  PROC DrawPart36()
    MoveL Offs(pOrigin,159.05,133.27,0.00),v40,z0,tPen\WObj:=wPaper;
    MoveL Offs(pOrigin,159.60,133.02,0.00),v40,z0,tPen\WObj:=wPaper;
    MoveL Offs(pOrigin,155.70,129.11,0.00),v40,z0,tPen\WObj:=wPaper;
    MoveL Offs(pOrigin,154.95,128.36,0.00),v40,z0,tPen\WObj:=wPaper;
    MoveL Offs(pOrigin,153.59,127.01,0.00),v40,z0,tPen\WObj:=wPaper;
    MoveL Offs(pOrigin,154.49,126.41,0.00),v40,z0,tPen\WObj:=wPaper;
    MoveL Offs(pOrigin,159.90,131.82,0.00),v40,z0,tPen\WObj:=wPaper;
    MoveL Offs(pOrigin,159.26,132.22,0.00),v40,z0,tPen\WObj:=wPaper;
    MoveL Offs(pOrigin,157.35,132.22,0.00),v40,z0,tPen\WObj:=wPaper;
    MoveL Offs(pOrigin,157.36,132.92,0.00),v40,z0,tPen\WObj:=wPaper;
    MoveL Offs(pOrigin,157.36,136.96,0.00),v40,z0,tPen\WObj:=wPaper;
    MoveL Offs(pOrigin,157.78,137.50,0.00),v40,z0,tPen\WObj:=wPaper;
    MoveL Offs(pOrigin,152.89,137.50,0.00),v40,z0,tPen\WObj:=wPaper;
    MoveL Offs(pOrigin,152.68,138.02,0.00),v40,z0,tPen\WObj:=wPaper;
    MoveL Offs(pOrigin,154.59,136.11,0.00),v40,z0,tPen\WObj:=wPaper;
    MoveL Offs(pOrigin,155.01,135.05,0.00),v40,z0,tPen\WObj:=wPaper;
    MoveL Offs(pOrigin,157.85,131.86,0.00),v40,z0,tPen\WObj:=wPaper;
    MoveL Offs(pOrigin,158.20,129.95,0.00),v40,z0,tPen\WObj:=wPaper;
    MoveL Offs(pOrigin,157.35,130.16,0.00),v40,z0,tPen\WObj:=wPaper;
    MoveL Offs(pOrigin,158.41,130.37,0.00),v40,z0,tPen\WObj:=wPaper;
    MoveL Offs(pOrigin,158.41,127.61,0.00),v40,z0,tPen\WObj:=wPaper;
    MoveL Offs(pOrigin,157.99,127.82,0.00),v40,z0,tPen\WObj:=wPaper;
    MoveL Offs(pOrigin,158.20,127.40,0.00),v40,z0,tPen\WObj:=wPaper;
    MoveL Offs(pOrigin,157.99,127.82,0.00),v40,z0,tPen\WObj:=wPaper;
    MoveL Offs(pOrigin,158.41,126.94,0.00),v40,z0,tPen\WObj:=wPaper;
    MoveL Offs(pOrigin,160.32,126.94,0.00),v40,z0,tPen\WObj:=wPaper;
    MoveL Offs(pOrigin,160.63,126.58,0.00),v40,z0,tPen\WObj:=wPaper;
    MoveL Offs(pOrigin,157.78,123.72,0.00),v40,z0,tPen\WObj:=wPaper;
    MoveL Offs(pOrigin,158.20,123.77,0.00),v40,z0,tPen\WObj:=wPaper;
    MoveL Offs(pOrigin,160.96,123.77,0.00),v40,z0,tPen\WObj:=wPaper;
    MoveL Offs(pOrigin,161.07,124.03,0.00),v40,z0,tPen\WObj:=wPaper;
    MoveL Offs(pOrigin,158.97,121.93,0.00),v40,z0,tPen\WObj:=wPaper;
    MoveL Offs(pOrigin,159.69,121.66,0.00),v40,z0,tPen\WObj:=wPaper;
    MoveL Offs(pOrigin,161.18,121.66,0.00),v40,z0,tPen\WObj:=wPaper;
    MoveL Offs(pOrigin,161.52,121.49,0.00),v40,z0,tPen\WObj:=wPaper;
    MoveL Offs(pOrigin,159.26,119.23,0.00),v40,z0,tPen\WObj:=wPaper;
    MoveL Offs(pOrigin,159.90,119.54,0.00),v40,z0,tPen\WObj:=wPaper;
    MoveL Offs(pOrigin,161.39,119.54,0.00),v40,z0,tPen\WObj:=wPaper;
    MoveL Offs(pOrigin,161.96,118.94,0.00),v40,z0,tPen\WObj:=wPaper;
    MoveL Offs(pOrigin,157.75,114.74,0.00),v40,z0,tPen\WObj:=wPaper;
    MoveL Offs(pOrigin,156.93,115.32,0.00),v40,z0,tPen\WObj:=wPaper;
    MoveL Offs(pOrigin,162.02,115.32,0.00),v40,z0,tPen\WObj:=wPaper;
    MoveL Offs(pOrigin,161.58,115.50,0.00),v40,z0,tPen\WObj:=wPaper;
    MoveL Offs(pOrigin,161.58,110.40,0.00),v40,z0,tPen\WObj:=wPaper;
    MoveL Offs(pOrigin,160.96,110.82,0.00),v40,z0,tPen\WObj:=wPaper;
    MoveL Offs(pOrigin,162.02,105.51,0.00),v40,z0,tPen\WObj:=wPaper;
    MoveL Offs(pOrigin,161.81,104.52,0.00),v40,z0,tPen\WObj:=wPaper;
    MoveL Offs(pOrigin,157.35,106.43,0.00),v40,z0,tPen\WObj:=wPaper;
    MoveL Offs(pOrigin,154.16,107.21,0.00),v40,z0,tPen\WObj:=wPaper;
    MoveL Offs(pOrigin,154.16,107.21,0.00),v40,z0,tPen\WObj:=wPaper;
    MoveL Offs(pOrigin,154.59,106.43,0.00),v40,z0,tPen\WObj:=wPaper;
    MoveL Offs(pOrigin,157.99,104.95,0.00),v40,z0,tPen\WObj:=wPaper;
    MoveL Offs(pOrigin,159.55,103.88,0.00),v40,z0,tPen\WObj:=wPaper;
    MoveL Offs(pOrigin,159.26,104.03,0.00),v40,z0,tPen\WObj:=wPaper;
    MoveL Offs(pOrigin,158.77,103.80,0.00),v40,z0,tPen\WObj:=wPaper;
    MoveL Offs(pOrigin,160.57,105.61,0.00),v40,z0,tPen\WObj:=wPaper;
    MoveL Offs(pOrigin,159.79,106.28,0.00),v40,z0,tPen\WObj:=wPaper;
    MoveL Offs(pOrigin,165.05,101.02,0.00),v40,z0,tPen\WObj:=wPaper;
    MoveL Offs(pOrigin,164.60,100.67,0.00),v40,z0,tPen\WObj:=wPaper;
    MoveL Offs(pOrigin,162.19,98.27,0.00),v40,z0,tPen\WObj:=wPaper;
    MoveL Offs(pOrigin,162.66,98.42,0.00),v40,z0,tPen\WObj:=wPaper;
    MoveL Offs(pOrigin,164.58,98.42,0.00),v40,z0,tPen\WObj:=wPaper;
    MoveL Offs(pOrigin,165.19,98.28,0.00),v40,z0,tPen\WObj:=wPaper;
    MoveL Offs(pOrigin,157.53,90.62,0.00),v40,z0,tPen\WObj:=wPaper;
    MoveL Offs(pOrigin,157.99,91.03,0.00),v40,z0,tPen\WObj:=wPaper;
    MoveL Offs(pOrigin,163.73,91.03,0.00),v40,z0,tPen\WObj:=wPaper;
    MoveL Offs(pOrigin,164.27,91.39,0.00),v40,z0,tPen\WObj:=wPaper;
    MoveL Offs(pOrigin,159.76,86.88,0.00),v40,z0,tPen\WObj:=wPaper;
    MoveL Offs(pOrigin,159.25,87.41,0.00),v40,z0,tPen\WObj:=wPaper;
    MoveL Offs(pOrigin,162.41,84.25,0.00),v40,z0,tPen\WObj:=wPaper;
    MoveL Offs(pOrigin,161.70,84.34,0.00),v40,z0,tPen\WObj:=wPaper;
    MoveL Offs(pOrigin,159.00,81.63,0.00),v40,z0,tPen\WObj:=wPaper;
    MoveL Offs(pOrigin,159.69,81.53,0.00),v40,z0,tPen\WObj:=wPaper;
    MoveL Offs(pOrigin,160.75,81.53,0.00),v40,z0,tPen\WObj:=wPaper;
    MoveL Offs(pOrigin,160.94,80.59,0.00),v40,z0,tPen\WObj:=wPaper;
    MoveL Offs(pOrigin,154.03,73.68,0.00),v40,fine,tPen\WObj:=wPaper;
    MoveL Offs(pOrigin,154.03,73.68,6.00),v60,z5,tPen\WObj:=wPaper;
    MoveL Offs(pOrigin,155.53,73.68,6.00),vTravel,z5,tPen\WObj:=wPaper;
    MoveL Offs(pOrigin,155.53,73.68,0.00),v60,z0,tPen\WObj:=wPaper;
    MoveL Offs(pOrigin,160.49,78.64,0.00),v40,z0,tPen\WObj:=wPaper;
    MoveL Offs(pOrigin,160.93,78.27,0.00),v40,z0,tPen\WObj:=wPaper;
    MoveL Offs(pOrigin,158.07,81.12,0.00),v40,z0,tPen\WObj:=wPaper;
    MoveL Offs(pOrigin,158.52,82.17,0.00),v40,z0,tPen\WObj:=wPaper;
    MoveL Offs(pOrigin,161.07,79.61,0.00),v40,z0,tPen\WObj:=wPaper;
    MoveL Offs(pOrigin,160.11,79.42,0.00),v40,z0,tPen\WObj:=wPaper;
    MoveL Offs(pOrigin,158.84,79.42,0.00),v40,z0,tPen\WObj:=wPaper;
    MoveL Offs(pOrigin,159.47,79.16,0.00),v40,z0,tPen\WObj:=wPaper;
    MoveL Offs(pOrigin,159.47,76.61,0.00),v40,z0,tPen\WObj:=wPaper;
    MoveL Offs(pOrigin,160.11,77.30,0.00),v40,z0,tPen\WObj:=wPaper;
    MoveL Offs(pOrigin,155.23,77.30,0.00),v40,z0,tPen\WObj:=wPaper;
    MoveL Offs(pOrigin,155.69,76.83,0.00),v40,z0,tPen\WObj:=wPaper;
    MoveL Offs(pOrigin,161.55,82.69,0.00),v40,z0,tPen\WObj:=wPaper;
    MoveL Offs(pOrigin,161.18,82.58,0.00),v40,z0,tPen\WObj:=wPaper;
    MoveL Offs(pOrigin,159.90,82.58,0.00),v40,z0,tPen\WObj:=wPaper;
    MoveL Offs(pOrigin,159.30,83.43,0.00),v40,z0,tPen\WObj:=wPaper;
    MoveL Offs(pOrigin,162.01,86.14,0.00),v40,z0,tPen\WObj:=wPaper;
    MoveL Offs(pOrigin,161.60,85.75,0.00),v40,z0,tPen\WObj:=wPaper;
    MoveL Offs(pOrigin,160.32,85.75,0.00),v40,z0,tPen\WObj:=wPaper;
    MoveL Offs(pOrigin,159.61,85.23,0.00),v40,z0,tPen\WObj:=wPaper;
    MoveL Offs(pOrigin,164.57,90.19,0.00),v40,z0,tPen\WObj:=wPaper;
    MoveL Offs(pOrigin,165.09,90.54,0.00),v40,z0,tPen\WObj:=wPaper;
    MoveL Offs(pOrigin,160.58,95.04,0.00),v40,z0,tPen\WObj:=wPaper;
    MoveL Offs(pOrigin,161.18,94.20,0.00),v40,z0,tPen\WObj:=wPaper;
    MoveL Offs(pOrigin,163.51,94.20,0.00),v40,z0,tPen\WObj:=wPaper;
    MoveL Offs(pOrigin,163.51,93.14,0.00),v40,z0,tPen\WObj:=wPaper;
    MoveL Offs(pOrigin,160.11,93.14,0.00),v40,z0,tPen\WObj:=wPaper;
    MoveL Offs(pOrigin,160.53,92.98,0.00),v40,z0,tPen\WObj:=wPaper;
    MoveL Offs(pOrigin,160.53,90.85,0.00),v40,z0,tPen\WObj:=wPaper;
    MoveL Offs(pOrigin,160.32,89.98,0.00),v40,z0,tPen\WObj:=wPaper;
    MoveL Offs(pOrigin,163.94,89.98,0.00),v40,fine,tPen\WObj:=wPaper;
    MoveL Offs(pOrigin,163.94,89.98,6.00),v60,z5,tPen\WObj:=wPaper;
    MoveL Offs(pOrigin,164.71,88.84,6.00),vTravel,z5,tPen\WObj:=wPaper;
    MoveL Offs(pOrigin,164.71,88.84,0.00),v60,z0,tPen\WObj:=wPaper;
    MoveL Offs(pOrigin,163.21,87.34,0.00),v40,z0,tPen\WObj:=wPaper;
    MoveL Offs(pOrigin,163.66,86.29,0.00),v40,z0,tPen\WObj:=wPaper;
    MoveL Offs(pOrigin,165.01,87.64,0.00),v40,z0,tPen\WObj:=wPaper;
    MoveL Offs(pOrigin,164.79,87.66,0.00),v40,z0,tPen\WObj:=wPaper;
    MoveL Offs(pOrigin,163.94,91.91,0.00),v40,z0,tPen\WObj:=wPaper;
    MoveL Offs(pOrigin,164.79,87.66,0.00),v40,z0,tPen\WObj:=wPaper;
    MoveL Offs(pOrigin,165.00,87.24,0.00),v40,z0,tPen\WObj:=wPaper;
  ENDPROC

  PROC DrawPart37()
    MoveL Offs(pOrigin,165.00,86.60,0.00),v40,z0,tPen\WObj:=wPaper;
    MoveL Offs(pOrigin,165.00,87.24,0.00),v40,z0,tPen\WObj:=wPaper;
    MoveL Offs(pOrigin,165.30,86.45,0.00),v40,z0,tPen\WObj:=wPaper;
    MoveL Offs(pOrigin,163.95,85.09,0.00),v40,fine,tPen\WObj:=wPaper;
    MoveL Offs(pOrigin,163.95,85.09,6.00),v60,z5,tPen\WObj:=wPaper;
    MoveL Offs(pOrigin,164.25,83.90,6.00),vTravel,z5,tPen\WObj:=wPaper;
    MoveL Offs(pOrigin,164.25,83.90,0.00),v60,z0,tPen\WObj:=wPaper;
    MoveL Offs(pOrigin,165.60,85.25,0.00),v40,z0,tPen\WObj:=wPaper;
    MoveL Offs(pOrigin,166.45,84.69,0.00),v40,z0,tPen\WObj:=wPaper;
    MoveL Offs(pOrigin,158.19,92.95,0.00),v40,z0,tPen\WObj:=wPaper;
    MoveL Offs(pOrigin,157.83,92.42,0.00),v40,z0,tPen\WObj:=wPaper;
    MoveL Offs(pOrigin,156.48,91.06,0.00),v40,z0,tPen\WObj:=wPaper;
    MoveL Offs(pOrigin,156.55,90.11,0.00),v40,z0,tPen\WObj:=wPaper;
    MoveL Offs(pOrigin,151.29,95.37,0.00),v40,z0,tPen\WObj:=wPaper;
    MoveL Offs(pOrigin,150.39,94.78,0.00),v40,z0,tPen\WObj:=wPaper;
    MoveL Offs(pOrigin,153.40,91.77,0.00),v40,z0,tPen\WObj:=wPaper;
    MoveL Offs(pOrigin,153.64,92.70,0.00),v40,z0,tPen\WObj:=wPaper;
    MoveL Offs(pOrigin,154.39,93.45,0.00),v40,z0,tPen\WObj:=wPaper;
    MoveL Offs(pOrigin,154.38,92.97,0.00),v40,z0,tPen\WObj:=wPaper;
    MoveL Offs(pOrigin,152.89,93.61,0.00),v40,z0,tPen\WObj:=wPaper;
    MoveL Offs(pOrigin,152.68,94.04,0.00),v40,z0,tPen\WObj:=wPaper;
    MoveL Offs(pOrigin,152.89,93.82,0.00),v40,z0,tPen\WObj:=wPaper;
    MoveL Offs(pOrigin,153.84,94.32,0.00),v40,z0,tPen\WObj:=wPaper;
    MoveL Offs(pOrigin,158.50,89.66,0.00),v40,z0,tPen\WObj:=wPaper;
    MoveL Offs(pOrigin,158.87,90.47,0.00),v40,z0,tPen\WObj:=wPaper;
    MoveL Offs(pOrigin,166.09,97.68,0.00),v40,z0,tPen\WObj:=wPaper;
    MoveL Offs(pOrigin,166.26,98.32,0.00),v40,z0,tPen\WObj:=wPaper;
    MoveL Offs(pOrigin,191.80,72.78,0.00),v40,z0,tPen\WObj:=wPaper;
    MoveL Offs(pOrigin,192.38,73.20,0.00),v40,z0,tPen\WObj:=wPaper;
    MoveL Offs(pOrigin,195.83,76.65,0.00),v40,z0,tPen\WObj:=wPaper;
    MoveL Offs(pOrigin,196.28,77.26,0.00),v40,z0,tPen\WObj:=wPaper;
    MoveL Offs(pOrigin,199.74,73.80,0.00),v40,z0,tPen\WObj:=wPaper;
    MoveL Offs(pOrigin,199.72,74.57,0.00),v40,z0,tPen\WObj:=wPaper;
    MoveL Offs(pOrigin,201.67,76.52,0.00),v40,z0,tPen\WObj:=wPaper;
    MoveL Offs(pOrigin,201.08,76.94,0.00),v40,z0,tPen\WObj:=wPaper;
    MoveL Offs(pOrigin,204.54,73.49,0.00),v40,z0,tPen\WObj:=wPaper;
    MoveL Offs(pOrigin,205.26,74.14,0.00),v40,z0,tPen\WObj:=wPaper;
    MoveL Offs(pOrigin,207.07,75.94,0.00),v40,z0,tPen\WObj:=wPaper;
    MoveL Offs(pOrigin,207.82,76.17,0.00),v40,z0,tPen\WObj:=wPaper;
    MoveL Offs(pOrigin,218.49,65.51,0.00),v40,z0,tPen\WObj:=wPaper;
    MoveL Offs(pOrigin,218.27,66.24,0.00),v40,z0,tPen\WObj:=wPaper;
    MoveL Offs(pOrigin,213.16,61.13,0.00),v40,z0,tPen\WObj:=wPaper;
    MoveL Offs(pOrigin,213.45,61.46,0.00),v40,z0,tPen\WObj:=wPaper;
    MoveL Offs(pOrigin,217.28,61.46,0.00),v40,z0,tPen\WObj:=wPaper;
    MoveL Offs(pOrigin,217.66,61.14,0.00),v40,z0,tPen\WObj:=wPaper;
    MoveL Offs(pOrigin,215.25,58.74,0.00),v40,z0,tPen\WObj:=wPaper;
    MoveL Offs(pOrigin,214.94,59.19,0.00),v40,z0,tPen\WObj:=wPaper;
    MoveL Offs(pOrigin,214.65,60.25,0.00),v40,z0,tPen\WObj:=wPaper;
    MoveL Offs(pOrigin,213.45,61.53,0.00),v40,z0,tPen\WObj:=wPaper;
    MoveL Offs(pOrigin,204.74,68.18,0.00),v40,z0,tPen\WObj:=wPaper;
    MoveL Offs(pOrigin,188.80,74.98,0.00),v40,z0,tPen\WObj:=wPaper;
    MoveL Offs(pOrigin,182.00,77.04,0.00),v40,z0,tPen\WObj:=wPaper;
    MoveL Offs(pOrigin,179.88,77.04,0.00),v40,z0,tPen\WObj:=wPaper;
    MoveL Offs(pOrigin,176.69,75.83,0.00),v40,z0,tPen\WObj:=wPaper;
    MoveL Offs(pOrigin,169.25,69.18,0.00),v40,z0,tPen\WObj:=wPaper;
    MoveL Offs(pOrigin,167.55,67.97,0.00),v40,z0,tPen\WObj:=wPaper;
    MoveL Offs(pOrigin,166.27,67.69,0.00),v40,z0,tPen\WObj:=wPaper;
    MoveL Offs(pOrigin,166.27,67.69,0.00),v40,z0,tPen\WObj:=wPaper;
    MoveL Offs(pOrigin,162.80,63.86,0.00),v40,z0,tPen\WObj:=wPaper;
    MoveL Offs(pOrigin,162.59,63.01,0.00),v40,z0,tPen\WObj:=wPaper;
    MoveL Offs(pOrigin,160.04,58.76,0.00),v40,z0,tPen\WObj:=wPaper;
    MoveL Offs(pOrigin,159.33,57.06,0.00),v40,z0,tPen\WObj:=wPaper;
    MoveL Offs(pOrigin,159.48,56.64,0.00),v40,fine,tPen\WObj:=wPaper;
    MoveL Offs(pOrigin,159.48,56.64,6.00),v60,z5,tPen\WObj:=wPaper;
    MoveL Offs(pOrigin,162.48,61.78,6.00),vTravel,z5,tPen\WObj:=wPaper;
    MoveL Offs(pOrigin,162.48,61.78,0.00),v60,z0,tPen\WObj:=wPaper;
    MoveL Offs(pOrigin,161.43,62.83,0.00),v40,z0,tPen\WObj:=wPaper;
    MoveL Offs(pOrigin,162.17,63.58,0.00),v40,z0,tPen\WObj:=wPaper;
    MoveL Offs(pOrigin,163.07,62.68,0.00),v40,z0,tPen\WObj:=wPaper;
    MoveL Offs(pOrigin,163.67,63.58,0.00),v40,z0,tPen\WObj:=wPaper;
    MoveL Offs(pOrigin,162.62,64.63,0.00),v40,z0,tPen\WObj:=wPaper;
    MoveL Offs(pOrigin,163.06,65.68,0.00),v40,z0,tPen\WObj:=wPaper;
    MoveL Offs(pOrigin,164.42,64.32,0.00),v40,z0,tPen\WObj:=wPaper;
    MoveL Offs(pOrigin,163.73,64.93,0.00),v40,z0,tPen\WObj:=wPaper;
    MoveL Offs(pOrigin,164.57,65.78,0.00),v40,z0,tPen\WObj:=wPaper;
    MoveL Offs(pOrigin,163.73,64.93,0.00),v40,fine,tPen\WObj:=wPaper;
    MoveL Offs(pOrigin,163.73,64.93,6.00),v60,z5,tPen\WObj:=wPaper;
    MoveL Offs(pOrigin,165.16,65.07,6.00),vTravel,z5,tPen\WObj:=wPaper;
    MoveL Offs(pOrigin,165.16,65.07,0.00),v60,z0,tPen\WObj:=wPaper;
    MoveL Offs(pOrigin,146.83,83.40,0.00),v40,z0,tPen\WObj:=wPaper;
    MoveL Offs(pOrigin,146.72,82.79,0.00),v40,z0,tPen\WObj:=wPaper;
    MoveL Offs(pOrigin,144.61,80.69,0.00),v40,z0,tPen\WObj:=wPaper;
    MoveL Offs(pOrigin,144.69,81.29,0.00),v40,z0,tPen\WObj:=wPaper;
    MoveL Offs(pOrigin,144.69,83.20,0.00),v40,z0,tPen\WObj:=wPaper;
    MoveL Offs(pOrigin,144.39,83.64,0.00),v40,z0,tPen\WObj:=wPaper;
    MoveL Offs(pOrigin,139.29,83.64,0.00),v40,fine,tPen\WObj:=wPaper;
    MoveL Offs(pOrigin,139.29,83.64,6.00),v60,z5,tPen\WObj:=wPaper;
    MoveL Offs(pOrigin,138.65,82.58,6.00),vTravel,z5,tPen\WObj:=wPaper;
    MoveL Offs(pOrigin,138.65,82.58,0.00),v60,z0,tPen\WObj:=wPaper;
    MoveL Offs(pOrigin,146.09,82.58,0.00),v40,z0,tPen\WObj:=wPaper;
    MoveL Offs(pOrigin,145.74,82.35,0.00),v40,z0,tPen\WObj:=wPaper;
    MoveL Offs(pOrigin,145.74,81.08,0.00),v40,z0,tPen\WObj:=wPaper;
    MoveL Offs(pOrigin,145.66,80.47,0.00),v40,z0,tPen\WObj:=wPaper;
    MoveL Offs(pOrigin,149.49,80.47,0.00),v40,z0,tPen\WObj:=wPaper;
    MoveL Offs(pOrigin,149.27,81.07,0.00),v40,z0,tPen\WObj:=wPaper;
    MoveL Offs(pOrigin,149.70,80.86,0.00),v40,z0,tPen\WObj:=wPaper;
    MoveL Offs(pOrigin,149.27,81.07,0.00),v40,z0,tPen\WObj:=wPaper;
    MoveL Offs(pOrigin,149.56,81.15,0.00),v40,z0,tPen\WObj:=wPaper;
    MoveL Offs(pOrigin,147.91,79.50,0.00),v40,z0,tPen\WObj:=wPaper;
    MoveL Offs(pOrigin,148.85,79.42,0.00),v40,z0,tPen\WObj:=wPaper;
    MoveL Offs(pOrigin,152.89,79.42,0.00),v40,z0,tPen\WObj:=wPaper;
    MoveL Offs(pOrigin,153.10,80.01,0.00),v40,z0,tPen\WObj:=wPaper;
    MoveL Offs(pOrigin,152.89,80.86,0.00),v40,z0,tPen\WObj:=wPaper;
    MoveL Offs(pOrigin,150.55,83.41,0.00),v40,z0,tPen\WObj:=wPaper;
    MoveL Offs(pOrigin,143.32,90.21,0.00),v40,z0,tPen\WObj:=wPaper;
    MoveL Offs(pOrigin,143.67,89.55,0.00),v40,z0,tPen\WObj:=wPaper;
    MoveL Offs(pOrigin,166.96,66.26,0.00),v40,z0,tPen\WObj:=wPaper;
    MoveL Offs(pOrigin,166.06,65.67,0.00),v40,z0,tPen\WObj:=wPaper;
    MoveL Offs(pOrigin,149.08,82.65,0.00),v40,z0,tPen\WObj:=wPaper;
    MoveL Offs(pOrigin,148.66,81.75,0.00),v40,z0,tPen\WObj:=wPaper;
    MoveL Offs(pOrigin,146.71,79.80,0.00),v40,z0,tPen\WObj:=wPaper;
    MoveL Offs(pOrigin,146.55,79.21,0.00),v40,z0,tPen\WObj:=wPaper;
    MoveL Offs(pOrigin,135.43,90.33,0.00),v40,z0,tPen\WObj:=wPaper;
    MoveL Offs(pOrigin,135.80,89.80,0.00),v40,z0,tPen\WObj:=wPaper;
    MoveL Offs(pOrigin,133.85,87.85,0.00),v40,z0,tPen\WObj:=wPaper;
    MoveL Offs(pOrigin,134.19,87.86,0.00),v40,z0,tPen\WObj:=wPaper;
    MoveL Offs(pOrigin,138.01,87.86,0.00),v40,z0,tPen\WObj:=wPaper;
    MoveL Offs(pOrigin,138.64,88.16,0.00),v40,z0,tPen\WObj:=wPaper;
    MoveL Offs(pOrigin,136.24,85.76,0.00),v40,z0,tPen\WObj:=wPaper;
    MoveL Offs(pOrigin,137.16,85.75,0.00),v40,z0,tPen\WObj:=wPaper;
  ENDPROC

  PROC DrawPart38()
    MoveL Offs(pOrigin,141.20,85.75,0.00),v40,z0,tPen\WObj:=wPaper;
    MoveL Offs(pOrigin,141.34,86.37,0.00),v40,z0,tPen\WObj:=wPaper;
    MoveL Offs(pOrigin,137.28,82.32,0.00),v40,z0,tPen\WObj:=wPaper;
    MoveL Offs(pOrigin,136.50,81.79,0.00),v40,z0,tPen\WObj:=wPaper;
    MoveL Offs(pOrigin,133.20,85.09,0.00),v40,z0,tPen\WObj:=wPaper;
    MoveL Offs(pOrigin,133.54,84.55,0.00),v40,z0,tPen\WObj:=wPaper;
    MoveL Offs(pOrigin,131.29,82.30,0.00),v40,z0,tPen\WObj:=wPaper;
    MoveL Offs(pOrigin,131.86,81.95,0.00),v40,z0,tPen\WObj:=wPaper;
    MoveL Offs(pOrigin,128.85,84.96,0.00),v40,z0,tPen\WObj:=wPaper;
    MoveL Offs(pOrigin,129.20,84.69,0.00),v40,z0,tPen\WObj:=wPaper;
    MoveL Offs(pOrigin,125.89,81.38,0.00),v40,z0,tPen\WObj:=wPaper;
    MoveL Offs(pOrigin,125.72,80.62,0.00),v40,z0,tPen\WObj:=wPaper;
    MoveL Offs(pOrigin,122.41,83.93,0.00),v40,z0,tPen\WObj:=wPaper;
    MoveL Offs(pOrigin,122.15,83.62,0.00),v40,z0,tPen\WObj:=wPaper;
    MoveL Offs(pOrigin,119.90,81.36,0.00),v40,fine,tPen\WObj:=wPaper;
    MoveL Offs(pOrigin,119.90,81.36,6.00),v60,z5,tPen\WObj:=wPaper;
    MoveL Offs(pOrigin,119.75,82.71,6.00),vTravel,z5,tPen\WObj:=wPaper;
    MoveL Offs(pOrigin,119.75,82.71,0.00),v60,z0,tPen\WObj:=wPaper;
    MoveL Offs(pOrigin,117.35,80.31,0.00),v40,z0,tPen\WObj:=wPaper;
    MoveL Offs(pOrigin,117.19,80.65,0.00),v40,z0,tPen\WObj:=wPaper;
    MoveL Offs(pOrigin,116.12,80.30,0.00),v40,z0,tPen\WObj:=wPaper;
    MoveL Offs(pOrigin,112.30,77.46,0.00),v40,z0,tPen\WObj:=wPaper;
    MoveL Offs(pOrigin,106.99,70.88,0.00),v40,z0,tPen\WObj:=wPaper;
    MoveL Offs(pOrigin,101.89,65.99,0.00),v40,z0,tPen\WObj:=wPaper;
    MoveL Offs(pOrigin,100.40,65.56,0.00),v40,z0,tPen\WObj:=wPaper;
    MoveL Offs(pOrigin,99.97,65.35,0.00),v40,z0,tPen\WObj:=wPaper;
    MoveL Offs(pOrigin,99.12,64.50,0.00),v40,z0,tPen\WObj:=wPaper;
    MoveL Offs(pOrigin,99.12,63.65,0.00),v40,z0,tPen\WObj:=wPaper;
    MoveL Offs(pOrigin,98.91,63.22,0.00),v40,z0,tPen\WObj:=wPaper;
    MoveL Offs(pOrigin,99.12,63.65,0.00),v40,z0,tPen\WObj:=wPaper;
    MoveL Offs(pOrigin,98.91,63.22,0.00),v40,fine,tPen\WObj:=wPaper;
    MoveL Offs(pOrigin,98.91,63.22,6.00),v60,z5,tPen\WObj:=wPaper;
    MoveL Offs(pOrigin,99.02,61.98,6.00),vTravel,z5,tPen\WObj:=wPaper;
    MoveL Offs(pOrigin,99.02,61.98,0.00),v60,z0,tPen\WObj:=wPaper;
    MoveL Offs(pOrigin,91.50,54.46,0.00),v40,z0,tPen\WObj:=wPaper;
    MoveL Offs(pOrigin,91.05,54.06,0.00),v40,z0,tPen\WObj:=wPaper;
    MoveL Offs(pOrigin,94.95,50.16,0.00),v40,z0,tPen\WObj:=wPaper;
    MoveL Offs(pOrigin,94.49,49.98,0.00),v40,z0,tPen\WObj:=wPaper;
    MoveL Offs(pOrigin,92.38,47.87,0.00),v40,z0,tPen\WObj:=wPaper;
    MoveL Offs(pOrigin,92.75,47.74,0.00),v40,z0,tPen\WObj:=wPaper;
    MoveL Offs(pOrigin,94.24,47.74,0.00),v40,z0,tPen\WObj:=wPaper;
    MoveL Offs(pOrigin,94.78,47.28,0.00),v40,z0,tPen\WObj:=wPaper;
    MoveL Offs(pOrigin,93.13,45.63,0.00),v40,z0,tPen\WObj:=wPaper;
    MoveL Offs(pOrigin,93.60,45.62,0.00),v40,z0,tPen\WObj:=wPaper;
    MoveL Offs(pOrigin,95.09,45.62,0.00),v40,z0,tPen\WObj:=wPaper;
    MoveL Offs(pOrigin,95.22,46.23,0.00),v40,z0,tPen\WObj:=wPaper;
    MoveL Offs(pOrigin,93.72,44.73,0.00),v40,z0,tPen\WObj:=wPaper;
    MoveL Offs(pOrigin,93.60,45.16,0.00),v40,z0,tPen\WObj:=wPaper;
    MoveL Offs(pOrigin,93.39,45.59,0.00),v40,z0,tPen\WObj:=wPaper;
    MoveL Offs(pOrigin,93.60,45.16,0.00),v40,z0,tPen\WObj:=wPaper;
    MoveL Offs(pOrigin,93.02,44.62,0.00),v40,z0,tPen\WObj:=wPaper;
    MoveL Offs(pOrigin,96.48,41.16,0.00),v40,z0,tPen\WObj:=wPaper;
    MoveL Offs(pOrigin,96.71,41.75,0.00),v40,z0,tPen\WObj:=wPaper;
    MoveL Offs(pOrigin,98.21,43.25,0.00),v40,z0,tPen\WObj:=wPaper;
    MoveL Offs(pOrigin,98.28,42.83,0.00),v40,z0,tPen\WObj:=wPaper;
    MoveL Offs(pOrigin,95.72,45.16,0.00),v40,z0,tPen\WObj:=wPaper;
    MoveL Offs(pOrigin,94.59,46.86,0.00),v40,z0,tPen\WObj:=wPaper;
    MoveL Offs(pOrigin,94.24,48.14,0.00),v40,z0,tPen\WObj:=wPaper;
    MoveL Offs(pOrigin,94.24,50.05,0.00),v40,z0,tPen\WObj:=wPaper;
    MoveL Offs(pOrigin,94.66,51.96,0.00),v40,z0,tPen\WObj:=wPaper;
    MoveL Offs(pOrigin,94.45,52.81,0.00),v40,z0,tPen\WObj:=wPaper;
    MoveL Offs(pOrigin,94.45,52.81,0.00),v40,z0,tPen\WObj:=wPaper;
    MoveL Offs(pOrigin,94.73,54.51,0.00),v40,z0,tPen\WObj:=wPaper;
    MoveL Offs(pOrigin,95.87,55.36,0.00),v40,z0,tPen\WObj:=wPaper;
    MoveL Offs(pOrigin,95.94,56.21,0.00),v40,z0,tPen\WObj:=wPaper;
    MoveL Offs(pOrigin,95.94,56.21,0.00),v40,z0,tPen\WObj:=wPaper;
    MoveL Offs(pOrigin,95.51,56.21,0.00),v40,z0,tPen\WObj:=wPaper;
    MoveL Offs(pOrigin,94.66,55.36,0.00),v40,z0,tPen\WObj:=wPaper;
    MoveL Offs(pOrigin,94.66,54.72,0.00),v40,z0,tPen\WObj:=wPaper;
    MoveL Offs(pOrigin,95.09,55.13,0.00),v40,z0,tPen\WObj:=wPaper;
    MoveL Offs(pOrigin,91.90,55.13,0.00),v40,z0,tPen\WObj:=wPaper;
    MoveL Offs(pOrigin,91.89,56.00,0.00),v40,z0,tPen\WObj:=wPaper;
    MoveL Offs(pOrigin,91.89,58.12,0.00),v40,z0,tPen\WObj:=wPaper;
    MoveL Offs(pOrigin,92.54,58.30,0.00),v40,z0,tPen\WObj:=wPaper;
    MoveL Offs(pOrigin,90.84,58.30,0.00),v40,z0,tPen\WObj:=wPaper;
    MoveL Offs(pOrigin,90.47,57.90,0.00),v40,z0,tPen\WObj:=wPaper;
    MoveL Offs(pOrigin,92.27,59.71,0.00),v40,z0,tPen\WObj:=wPaper;
    MoveL Offs(pOrigin,91.90,59.35,0.00),v40,z0,tPen\WObj:=wPaper;
    MoveL Offs(pOrigin,90.41,59.35,0.00),v40,z0,tPen\WObj:=wPaper;
    MoveL Offs(pOrigin,90.02,58.95,0.00),v40,z0,tPen\WObj:=wPaper;
    MoveL Offs(pOrigin,91.97,60.91,0.00),v40,z0,tPen\WObj:=wPaper;
    MoveL Offs(pOrigin,91.69,60.41,0.00),v40,z0,tPen\WObj:=wPaper;
    MoveL Offs(pOrigin,90.20,60.41,0.00),v40,z0,tPen\WObj:=wPaper;
    MoveL Offs(pOrigin,89.87,60.30,0.00),v40,z0,tPen\WObj:=wPaper;
    MoveL Offs(pOrigin,91.68,62.10,0.00),v40,z0,tPen\WObj:=wPaper;
    MoveL Offs(pOrigin,91.26,62.52,0.00),v40,z0,tPen\WObj:=wPaper;
    MoveL Offs(pOrigin,89.78,62.52,0.00),v40,z0,tPen\WObj:=wPaper;
    MoveL Offs(pOrigin,89.28,62.69,0.00),v40,z0,tPen\WObj:=wPaper;
    MoveL Offs(pOrigin,91.24,64.65,0.00),v40,z0,tPen\WObj:=wPaper;
    MoveL Offs(pOrigin,90.84,64.63,0.00),v40,z0,tPen\WObj:=wPaper;
    MoveL Offs(pOrigin,89.35,64.63,0.00),v40,z0,tPen\WObj:=wPaper;
    MoveL Offs(pOrigin,88.84,65.24,0.00),v40,z0,tPen\WObj:=wPaper;
    MoveL Offs(pOrigin,91.25,67.64,0.00),v40,z0,tPen\WObj:=wPaper;
    MoveL Offs(pOrigin,90.84,67.80,0.00),v40,z0,tPen\WObj:=wPaper;
    MoveL Offs(pOrigin,89.14,67.80,0.00),v40,z0,tPen\WObj:=wPaper;
    MoveL Offs(pOrigin,88.55,67.94,0.00),v40,z0,tPen\WObj:=wPaper;
    MoveL Offs(pOrigin,91.40,70.79,0.00),v40,z0,tPen\WObj:=wPaper;
    MoveL Offs(pOrigin,91.05,70.97,0.00),v40,z0,tPen\WObj:=wPaper;
    MoveL Offs(pOrigin,89.56,70.97,0.00),v40,z0,tPen\WObj:=wPaper;
    MoveL Offs(pOrigin,89.01,71.38,0.00),v40,z0,tPen\WObj:=wPaper;
    MoveL Offs(pOrigin,93.37,75.74,0.00),v40,z0,tPen\WObj:=wPaper;
    MoveL Offs(pOrigin,93.53,75.48,0.00),v40,z0,tPen\WObj:=wPaper;
    MoveL Offs(pOrigin,91.12,77.88,0.00),v40,z0,tPen\WObj:=wPaper;
    MoveL Offs(pOrigin,91.69,77.04,0.00),v40,z0,tPen\WObj:=wPaper;
    MoveL Offs(pOrigin,91.90,77.46,0.00),v40,z0,tPen\WObj:=wPaper;
    MoveL Offs(pOrigin,91.69,77.04,0.00),v40,z0,tPen\WObj:=wPaper;
    MoveL Offs(pOrigin,92.11,77.30,0.00),v40,z0,tPen\WObj:=wPaper;
    MoveL Offs(pOrigin,93.81,77.30,0.00),v40,z0,tPen\WObj:=wPaper;
    MoveL Offs(pOrigin,93.39,76.82,0.00),v40,z0,tPen\WObj:=wPaper;
    MoveL Offs(pOrigin,93.81,77.46,0.00),v40,z0,tPen\WObj:=wPaper;
    MoveL Offs(pOrigin,93.39,76.82,0.00),v40,z0,tPen\WObj:=wPaper;
    MoveL Offs(pOrigin,93.18,76.25,0.00),v40,z0,tPen\WObj:=wPaper;
    MoveL Offs(pOrigin,91.48,76.25,0.00),v40,z0,tPen\WObj:=wPaper;
    MoveL Offs(pOrigin,91.26,76.19,0.00),v40,z0,tPen\WObj:=wPaper;
    MoveL Offs(pOrigin,91.47,76.61,0.00),v40,z0,tPen\WObj:=wPaper;
    MoveL Offs(pOrigin,91.26,76.19,0.00),v40,z0,tPen\WObj:=wPaper;
    MoveL Offs(pOrigin,90.83,76.68,0.00),v40,z0,tPen\WObj:=wPaper;
    MoveL Offs(pOrigin,93.23,74.28,0.00),v40,z0,tPen\WObj:=wPaper;
    MoveL Offs(pOrigin,92.75,75.19,0.00),v40,z0,tPen\WObj:=wPaper;
    MoveL Offs(pOrigin,91.05,75.19,0.00),v40,z0,tPen\WObj:=wPaper;
  ENDPROC

  PROC DrawPart39()
    MoveL Offs(pOrigin,90.52,75.88,0.00),v40,z0,tPen\WObj:=wPaper;
    MoveL Offs(pOrigin,97.43,82.79,0.00),v40,z0,tPen\WObj:=wPaper;
    MoveL Offs(pOrigin,97.00,82.58,0.00),v40,z0,tPen\WObj:=wPaper;
    MoveL Offs(pOrigin,95.30,82.58,0.00),v40,z0,tPen\WObj:=wPaper;
    MoveL Offs(pOrigin,94.88,82.35,0.00),v40,z0,tPen\WObj:=wPaper;
    MoveL Offs(pOrigin,95.09,82.78,0.00),v40,z0,tPen\WObj:=wPaper;
    MoveL Offs(pOrigin,94.88,82.35,0.00),v40,z0,tPen\WObj:=wPaper;
    MoveL Offs(pOrigin,94.74,83.08,0.00),v40,z0,tPen\WObj:=wPaper;
    MoveL Offs(pOrigin,99.55,87.89,0.00),v40,z0,tPen\WObj:=wPaper;
    MoveL Offs(pOrigin,99.63,87.29,0.00),v40,z0,tPen\WObj:=wPaper;
    MoveL Offs(pOrigin,97.23,89.70,0.00),v40,z0,tPen\WObj:=wPaper;
    MoveL Offs(pOrigin,98.06,89.57,0.00),v40,z0,tPen\WObj:=wPaper;
    MoveL Offs(pOrigin,98.28,90.00,0.00),v40,z0,tPen\WObj:=wPaper;
    MoveL Offs(pOrigin,98.06,89.57,0.00),v40,z0,tPen\WObj:=wPaper;
    MoveL Offs(pOrigin,98.06,88.92,0.00),v40,z0,tPen\WObj:=wPaper;
    MoveL Offs(pOrigin,99.55,88.92,0.00),v40,z0,tPen\WObj:=wPaper;
    MoveL Offs(pOrigin,99.76,89.36,0.00),v40,z0,tPen\WObj:=wPaper;
    MoveL Offs(pOrigin,100.19,89.79,0.00),v40,z0,tPen\WObj:=wPaper;
    MoveL Offs(pOrigin,99.76,89.36,0.00),v40,z0,tPen\WObj:=wPaper;
    MoveL Offs(pOrigin,100.40,89.98,0.00),v40,z0,tPen\WObj:=wPaper;
    MoveL Offs(pOrigin,98.70,89.98,0.00),v40,z0,tPen\WObj:=wPaper;
    MoveL Offs(pOrigin,97.83,90.59,0.00),v40,z0,tPen\WObj:=wPaper;
    MoveL Offs(pOrigin,100.08,88.34,0.00),v40,z0,tPen\WObj:=wPaper;
    MoveL Offs(pOrigin,100.68,89.24,0.00),v40,z0,tPen\WObj:=wPaper;
    MoveL Offs(pOrigin,98.57,91.34,0.00),v40,z0,tPen\WObj:=wPaper;
    MoveL Offs(pOrigin,99.34,91.03,0.00),v40,z0,tPen\WObj:=wPaper;
    MoveL Offs(pOrigin,101.25,91.03,0.00),v40,z0,tPen\WObj:=wPaper;
    MoveL Offs(pOrigin,102.17,90.73,0.00),v40,z0,tPen\WObj:=wPaper;
    MoveL Offs(pOrigin,100.07,92.83,0.00),v40,z0,tPen\WObj:=wPaper;
    MoveL Offs(pOrigin,99.97,92.12,0.00),v40,z0,tPen\WObj:=wPaper;
    MoveL Offs(pOrigin,101.25,93.19,0.00),v40,z0,tPen\WObj:=wPaper;
    MoveL Offs(pOrigin,99.97,92.12,0.00),v40,z0,tPen\WObj:=wPaper;
    MoveL Offs(pOrigin,100.40,92.09,0.00),v40,z0,tPen\WObj:=wPaper;
    MoveL Offs(pOrigin,102.52,92.09,0.00),v40,z0,tPen\WObj:=wPaper;
    MoveL Offs(pOrigin,102.53,92.12,0.00),v40,z0,tPen\WObj:=wPaper;
    MoveL Offs(pOrigin,102.95,92.55,0.00),v40,z0,tPen\WObj:=wPaper;
    MoveL Offs(pOrigin,102.53,92.12,0.00),v40,z0,tPen\WObj:=wPaper;
    MoveL Offs(pOrigin,103.07,91.33,0.00),v40,z0,tPen\WObj:=wPaper;
    MoveL Offs(pOrigin,100.81,93.58,0.00),v40,z0,tPen\WObj:=wPaper;
    MoveL Offs(pOrigin,101.68,93.14,0.00),v40,z0,tPen\WObj:=wPaper;
    MoveL Offs(pOrigin,104.01,93.14,0.00),v40,z0,tPen\WObj:=wPaper;
    MoveL Offs(pOrigin,103.50,93.61,0.00),v40,z0,tPen\WObj:=wPaper;
    MoveL Offs(pOrigin,103.50,95.31,0.00),v40,z0,tPen\WObj:=wPaper;
    MoveL Offs(pOrigin,103.16,95.26,0.00),v40,z0,tPen\WObj:=wPaper;
    MoveL Offs(pOrigin,106.99,95.26,0.00),v40,z0,tPen\WObj:=wPaper;
    MoveL Offs(pOrigin,107.40,94.46,0.00),v40,z0,tPen\WObj:=wPaper;
    MoveL Offs(pOrigin,103.34,98.52,0.00),v40,z0,tPen\WObj:=wPaper;
    MoveL Offs(pOrigin,103.47,97.79,0.00),v40,z0,tPen\WObj:=wPaper;
    MoveL Offs(pOrigin,107.38,101.70,0.00),v40,z0,tPen\WObj:=wPaper;
    MoveL Offs(pOrigin,106.56,101.59,0.00),v40,z0,tPen\WObj:=wPaper;
    MoveL Offs(pOrigin,105.29,101.59,0.00),v40,z0,tPen\WObj:=wPaper;
    MoveL Offs(pOrigin,104.83,102.14,0.00),v40,z0,tPen\WObj:=wPaper;
    MoveL Offs(pOrigin,108.74,106.05,0.00),v40,z0,tPen\WObj:=wPaper;
    MoveL Offs(pOrigin,108.05,105.82,0.00),v40,z0,tPen\WObj:=wPaper;
    MoveL Offs(pOrigin,106.78,105.82,0.00),v40,z0,tPen\WObj:=wPaper;
    MoveL Offs(pOrigin,106.34,106.64,0.00),v40,z0,tPen\WObj:=wPaper;
    MoveL Offs(pOrigin,116.41,116.71,0.00),v40,z0,tPen\WObj:=wPaper;
    MoveL Offs(pOrigin,116.62,116.60,0.00),v40,z0,tPen\WObj:=wPaper;
    MoveL Offs(pOrigin,114.37,118.85,0.00),v40,z0,tPen\WObj:=wPaper;
    MoveL Offs(pOrigin,114.85,118.26,0.00),v40,z0,tPen\WObj:=wPaper;
    MoveL Offs(pOrigin,115.06,118.69,0.00),v40,z0,tPen\WObj:=wPaper;
    MoveL Offs(pOrigin,114.85,118.26,0.00),v40,z0,tPen\WObj:=wPaper;
    MoveL Offs(pOrigin,115.49,118.49,0.00),v40,z0,tPen\WObj:=wPaper;
    MoveL Offs(pOrigin,116.76,118.49,0.00),v40,z0,tPen\WObj:=wPaper;
    MoveL Offs(pOrigin,116.76,118.05,0.00),v40,z0,tPen\WObj:=wPaper;
    MoveL Offs(pOrigin,116.97,118.47,0.00),v40,z0,tPen\WObj:=wPaper;
    MoveL Offs(pOrigin,116.76,118.05,0.00),v40,z0,tPen\WObj:=wPaper;
    MoveL Offs(pOrigin,117.22,117.50,0.00),v40,z0,tPen\WObj:=wPaper;
    MoveL Offs(pOrigin,114.96,119.75,0.00),v40,z0,tPen\WObj:=wPaper;
    MoveL Offs(pOrigin,115.37,120.15,0.00),v40,z0,tPen\WObj:=wPaper;
    MoveL Offs(pOrigin,118.38,123.15,0.00),v40,z0,tPen\WObj:=wPaper;
    MoveL Offs(pOrigin,118.04,122.71,0.00),v40,z0,tPen\WObj:=wPaper;
    MoveL Offs(pOrigin,116.76,122.71,0.00),v40,z0,tPen\WObj:=wPaper;
    MoveL Offs(pOrigin,115.98,122.25,0.00),v40,z0,tPen\WObj:=wPaper;
    MoveL Offs(pOrigin,118.83,125.10,0.00),v40,z0,tPen\WObj:=wPaper;
    MoveL Offs(pOrigin,118.25,124.82,0.00),v40,z0,tPen\WObj:=wPaper;
    MoveL Offs(pOrigin,117.19,124.82,0.00),v40,z0,tPen\WObj:=wPaper;
    MoveL Offs(pOrigin,116.44,124.20,0.00),v40,z0,tPen\WObj:=wPaper;
    MoveL Offs(pOrigin,118.99,126.75,0.00),v40,z0,tPen\WObj:=wPaper;
    MoveL Offs(pOrigin,118.68,126.94,0.00),v40,z0,tPen\WObj:=wPaper;
    MoveL Offs(pOrigin,117.40,126.94,0.00),v40,z0,tPen\WObj:=wPaper;
    MoveL Offs(pOrigin,116.75,127.49,0.00),v40,z0,tPen\WObj:=wPaper;
    MoveL Offs(pOrigin,125.16,135.91,0.00),v40,z0,tPen\WObj:=wPaper;
    MoveL Offs(pOrigin,125.70,135.90,0.00),v40,z0,tPen\WObj:=wPaper;
    MoveL Offs(pOrigin,123.60,138.00,0.00),v40,z0,tPen\WObj:=wPaper;
    MoveL Offs(pOrigin,124.41,137.50,0.00),v40,z0,tPen\WObj:=wPaper;
    MoveL Offs(pOrigin,125.90,137.50,0.00),v40,z0,tPen\WObj:=wPaper;
    MoveL Offs(pOrigin,125.69,137.18,0.00),v40,z0,tPen\WObj:=wPaper;
    MoveL Offs(pOrigin,126.75,138.24,0.00),v40,z0,tPen\WObj:=wPaper;
    MoveL Offs(pOrigin,125.69,137.18,0.00),v40,z0,tPen\WObj:=wPaper;
    MoveL Offs(pOrigin,126.45,136.64,0.00),v40,z0,tPen\WObj:=wPaper;
    MoveL Offs(pOrigin,124.19,138.90,0.00),v40,z0,tPen\WObj:=wPaper;
    MoveL Offs(pOrigin,124.94,139.64,0.00),v40,z0,tPen\WObj:=wPaper;
    MoveL Offs(pOrigin,127.19,137.39,0.00),v40,z0,tPen\WObj:=wPaper;
    MoveL Offs(pOrigin,127.64,138.44,0.00),v40,z0,tPen\WObj:=wPaper;
    MoveL Offs(pOrigin,125.23,140.84,0.00),v40,z0,tPen\WObj:=wPaper;
    MoveL Offs(pOrigin,125.47,140.70,0.00),v40,z0,tPen\WObj:=wPaper;
    MoveL Offs(pOrigin,127.88,143.11,0.00),v40,z0,tPen\WObj:=wPaper;
    MoveL Offs(pOrigin,127.60,142.78,0.00),v40,z0,tPen\WObj:=wPaper;
    MoveL Offs(pOrigin,126.54,142.78,0.00),v40,z0,tPen\WObj:=wPaper;
    MoveL Offs(pOrigin,125.78,142.50,0.00),v40,z0,tPen\WObj:=wPaper;
    MoveL Offs(pOrigin,127.88,144.60,0.00),v40,z0,tPen\WObj:=wPaper;
    MoveL Offs(pOrigin,127.60,144.89,0.00),v40,z0,tPen\WObj:=wPaper;
    MoveL Offs(pOrigin,126.32,144.89,0.00),v40,z0,tPen\WObj:=wPaper;
    MoveL Offs(pOrigin,125.79,145.50,0.00),v40,z0,tPen\WObj:=wPaper;
    MoveL Offs(pOrigin,130.90,150.60,0.00),v40,z0,tPen\WObj:=wPaper;
    MoveL Offs(pOrigin,130.79,151.22,0.00),v40,z0,tPen\WObj:=wPaper;
    MoveL Offs(pOrigin,129.72,151.22,0.00),v40,z0,tPen\WObj:=wPaper;
    MoveL Offs(pOrigin,128.95,151.65,0.00),v40,z0,tPen\WObj:=wPaper;
    MoveL Offs(pOrigin,131.21,153.90,0.00),v40,z0,tPen\WObj:=wPaper;
    MoveL Offs(pOrigin,131.79,153.70,0.00),v40,z0,tPen\WObj:=wPaper;
    MoveL Offs(pOrigin,128.78,156.71,0.00),v40,z0,tPen\WObj:=wPaper;
    MoveL Offs(pOrigin,129.27,156.44,0.00),v40,z0,tPen\WObj:=wPaper;
    MoveL Offs(pOrigin,134.53,161.70,0.00),v40,z0,tPen\WObj:=wPaper;
    MoveL Offs(pOrigin,134.19,161.78,0.00),v40,z0,tPen\WObj:=wPaper;
    MoveL Offs(pOrigin,133.12,161.78,0.00),v40,z0,tPen\WObj:=wPaper;
    MoveL Offs(pOrigin,133.12,162.84,0.00),v40,z0,tPen\WObj:=wPaper;
    MoveL Offs(pOrigin,134.19,162.84,0.00),v40,z0,tPen\WObj:=wPaper;
    MoveL Offs(pOrigin,134.53,163.20,0.00),v40,z0,tPen\WObj:=wPaper;
    MoveL Offs(pOrigin,130.02,158.69,0.00),v40,z0,tPen\WObj:=wPaper;
  ENDPROC

  PROC DrawPart40()
    MoveL Offs(pOrigin,129.67,158.80,0.00),v40,z0,tPen\WObj:=wPaper;
    MoveL Offs(pOrigin,131.93,156.55,0.00),v40,z0,tPen\WObj:=wPaper;
    MoveL Offs(pOrigin,131.00,156.50,0.00),v40,z0,tPen\WObj:=wPaper;
    MoveL Offs(pOrigin,129.94,156.50,0.00),v40,z0,tPen\WObj:=wPaper;
    MoveL Offs(pOrigin,130.15,157.56,0.00),v40,z0,tPen\WObj:=wPaper;
    MoveL Offs(pOrigin,131.43,157.56,0.00),v40,z0,tPen\WObj:=wPaper;
    MoveL Offs(pOrigin,131.85,158.00,0.00),v40,z0,tPen\WObj:=wPaper;
    MoveL Offs(pOrigin,132.27,158.43,0.00),v40,z0,tPen\WObj:=wPaper;
    MoveL Offs(pOrigin,131.85,158.00,0.00),v40,z0,tPen\WObj:=wPaper;
    MoveL Offs(pOrigin,132.52,157.45,0.00),v40,z0,tPen\WObj:=wPaper;
    MoveL Offs(pOrigin,130.42,159.55,0.00),v40,z0,tPen\WObj:=wPaper;
    MoveL Offs(pOrigin,130.57,159.06,0.00),v40,z0,tPen\WObj:=wPaper;
    MoveL Offs(pOrigin,131.21,159.70,0.00),v40,z0,tPen\WObj:=wPaper;
    MoveL Offs(pOrigin,130.57,159.06,0.00),v40,z0,tPen\WObj:=wPaper;
    MoveL Offs(pOrigin,130.79,158.62,0.00),v40,z0,tPen\WObj:=wPaper;
    MoveL Offs(pOrigin,132.49,158.62,0.00),v40,z0,tPen\WObj:=wPaper;
    MoveL Offs(pOrigin,133.12,159.06,0.00),v40,z0,tPen\WObj:=wPaper;
    MoveL Offs(pOrigin,133.55,159.27,0.00),v40,z0,tPen\WObj:=wPaper;
    MoveL Offs(pOrigin,133.12,159.06,0.00),v40,z0,tPen\WObj:=wPaper;
    MoveL Offs(pOrigin,133.55,159.67,0.00),v40,z0,tPen\WObj:=wPaper;
    MoveL Offs(pOrigin,131.85,159.67,0.00),v40,z0,tPen\WObj:=wPaper;
    MoveL Offs(pOrigin,131.02,160.45,0.00),v40,z0,tPen\WObj:=wPaper;
    MoveL Offs(pOrigin,133.42,158.04,0.00),v40,z0,tPen\WObj:=wPaper;
    MoveL Offs(pOrigin,134.02,158.94,0.00),v40,z0,tPen\WObj:=wPaper;
    MoveL Offs(pOrigin,131.61,161.34,0.00),v40,fine,tPen\WObj:=wPaper;
    MoveL Offs(pOrigin,131.61,161.34,6.00),v60,z5,tPen\WObj:=wPaper;
    MoveL Offs(pOrigin,131.91,162.54,6.00),vTravel,z5,tPen\WObj:=wPaper;
    MoveL Offs(pOrigin,131.91,162.54,0.00),v60,z0,tPen\WObj:=wPaper;
    MoveL Offs(pOrigin,134.76,159.69,0.00),v40,z0,tPen\WObj:=wPaper;
    MoveL Offs(pOrigin,134.07,159.75,0.00),v40,z0,tPen\WObj:=wPaper;
    MoveL Offs(pOrigin,129.26,154.94,0.00),v40,z0,tPen\WObj:=wPaper;
    MoveL Offs(pOrigin,129.72,155.45,0.00),v40,z0,tPen\WObj:=wPaper;
    MoveL Offs(pOrigin,130.79,155.45,0.00),v40,z0,tPen\WObj:=wPaper;
    MoveL Offs(pOrigin,131.21,155.40,0.00),v40,z0,tPen\WObj:=wPaper;
    MoveL Offs(pOrigin,129.26,153.45,0.00),v40,z0,tPen\WObj:=wPaper;
    MoveL Offs(pOrigin,129.72,153.34,0.00),v40,z0,tPen\WObj:=wPaper;
    MoveL Offs(pOrigin,130.79,153.34,0.00),v40,z0,tPen\WObj:=wPaper;
    MoveL Offs(pOrigin,131.35,152.55,0.00),v40,z0,tPen\WObj:=wPaper;
    MoveL Offs(pOrigin,126.24,147.44,0.00),v40,z0,tPen\WObj:=wPaper;
    MoveL Offs(pOrigin,125.81,147.73,0.00),v40,z0,tPen\WObj:=wPaper;
    MoveL Offs(pOrigin,128.37,145.18,0.00),v40,z0,tPen\WObj:=wPaper;
    MoveL Offs(pOrigin,127.60,145.94,0.00),v40,z0,tPen\WObj:=wPaper;
    MoveL Offs(pOrigin,126.54,145.94,0.00),v40,z0,tPen\WObj:=wPaper;
    MoveL Offs(pOrigin,126.75,147.00,0.00),v40,z0,tPen\WObj:=wPaper;
    MoveL Offs(pOrigin,128.02,147.00,0.00),v40,z0,tPen\WObj:=wPaper;
    MoveL Offs(pOrigin,128.02,146.95,0.00),v40,z0,tPen\WObj:=wPaper;
    MoveL Offs(pOrigin,128.24,147.38,0.00),v40,z0,tPen\WObj:=wPaper;
    MoveL Offs(pOrigin,128.02,146.95,0.00),v40,z0,tPen\WObj:=wPaper;
    MoveL Offs(pOrigin,128.19,146.40,0.00),v40,z0,tPen\WObj:=wPaper;
    MoveL Offs(pOrigin,125.78,144.00,0.00),v40,z0,tPen\WObj:=wPaper;
    MoveL Offs(pOrigin,125.38,143.69,0.00),v40,z0,tPen\WObj:=wPaper;
    MoveL Offs(pOrigin,128.38,140.68,0.00),v40,z0,tPen\WObj:=wPaper;
    MoveL Offs(pOrigin,127.60,140.66,0.00),v40,z0,tPen\WObj:=wPaper;
    MoveL Offs(pOrigin,126.32,140.66,0.00),v40,z0,tPen\WObj:=wPaper;
    MoveL Offs(pOrigin,126.54,141.72,0.00),v40,z0,tPen\WObj:=wPaper;
    MoveL Offs(pOrigin,127.60,141.72,0.00),v40,z0,tPen\WObj:=wPaper;
    MoveL Offs(pOrigin,127.87,141.61,0.00),v40,z0,tPen\WObj:=wPaper;
    MoveL Offs(pOrigin,123.22,136.95,0.00),v40,z0,tPen\WObj:=wPaper;
    MoveL Offs(pOrigin,123.15,136.95,0.00),v40,z0,tPen\WObj:=wPaper;
    MoveL Offs(pOrigin,129.16,130.94,0.00),v40,z0,tPen\WObj:=wPaper;
    MoveL Offs(pOrigin,129.64,131.43,0.00),v40,z0,tPen\WObj:=wPaper;
    MoveL Offs(pOrigin,131.14,132.93,0.00),v40,z0,tPen\WObj:=wPaper;
    MoveL Offs(pOrigin,131.25,133.33,0.00),v40,z0,tPen\WObj:=wPaper;
    MoveL Offs(pOrigin,134.71,129.88,0.00),v40,z0,tPen\WObj:=wPaper;
    MoveL Offs(pOrigin,134.73,130.54,0.00),v40,z0,tPen\WObj:=wPaper;
    MoveL Offs(pOrigin,136.08,131.90,0.00),v40,z0,tPen\WObj:=wPaper;
    MoveL Offs(pOrigin,136.80,132.27,0.00),v40,z0,tPen\WObj:=wPaper;
    MoveL Offs(pOrigin,140.70,128.36,0.00),v40,z0,tPen\WObj:=wPaper;
    MoveL Offs(pOrigin,140.72,129.06,0.00),v40,z0,tPen\WObj:=wPaper;
    MoveL Offs(pOrigin,142.07,130.42,0.00),v40,z0,tPen\WObj:=wPaper;
    MoveL Offs(pOrigin,143.12,129.97,0.00),v40,z0,tPen\WObj:=wPaper;
    MoveL Offs(pOrigin,141.76,128.62,0.00),v40,fine,tPen\WObj:=wPaper;
    MoveL Offs(pOrigin,141.76,128.62,6.00),v60,z5,tPen\WObj:=wPaper;
    MoveL Offs(pOrigin,142.80,127.76,6.00),vTravel,z5,tPen\WObj:=wPaper;
    MoveL Offs(pOrigin,142.80,127.76,0.00),v60,z0,tPen\WObj:=wPaper;
    MoveL Offs(pOrigin,138.74,131.81,0.00),v40,z0,tPen\WObj:=wPaper;
    MoveL Offs(pOrigin,138.48,131.30,0.00),v40,z0,tPen\WObj:=wPaper;
    MoveL Offs(pOrigin,137.13,129.95,0.00),v40,z0,tPen\WObj:=wPaper;
    MoveL Offs(pOrigin,136.65,129.42,0.00),v40,z0,tPen\WObj:=wPaper;
    MoveL Offs(pOrigin,132.90,133.18,0.00),v40,z0,tPen\WObj:=wPaper;
    MoveL Offs(pOrigin,132.34,132.63,0.00),v40,z0,tPen\WObj:=wPaper;
    MoveL Offs(pOrigin,130.84,131.13,0.00),v40,z0,tPen\WObj:=wPaper;
    MoveL Offs(pOrigin,131.11,130.49,0.00),v40,z0,tPen\WObj:=wPaper;
    MoveL Offs(pOrigin,127.65,133.94,0.00),v40,z0,tPen\WObj:=wPaper;
    MoveL Offs(pOrigin,127.25,133.52,0.00),v40,z0,tPen\WObj:=wPaper;
    MoveL Offs(pOrigin,125.75,132.01,0.00),v40,z0,tPen\WObj:=wPaper;
    MoveL Offs(pOrigin,126.01,131.10,0.00),v40,z0,tPen\WObj:=wPaper;
    MoveL Offs(pOrigin,122.26,134.86,0.00),v40,z0,tPen\WObj:=wPaper;
    MoveL Offs(pOrigin,123.14,134.33,0.00),v40,z0,tPen\WObj:=wPaper;
    MoveL Offs(pOrigin,124.62,134.33,0.00),v40,z0,tPen\WObj:=wPaper;
    MoveL Offs(pOrigin,125.15,134.41,0.00),v40,z0,tPen\WObj:=wPaper;
    MoveL Offs(pOrigin,122.75,132.00,0.00),v40,z0,tPen\WObj:=wPaper;
    MoveL Offs(pOrigin,122.72,131.41,0.00),v40,z0,tPen\WObj:=wPaper;
    MoveL Offs(pOrigin,120.31,133.82,0.00),v40,z0,tPen\WObj:=wPaper;
    MoveL Offs(pOrigin,119.95,132.93,0.00),v40,z0,tPen\WObj:=wPaper;
    MoveL Offs(pOrigin,120.38,133.14,0.00),v40,z0,tPen\WObj:=wPaper;
    MoveL Offs(pOrigin,119.95,132.93,0.00),v40,z0,tPen\WObj:=wPaper;
    MoveL Offs(pOrigin,119.42,133.22,0.00),v40,z0,tPen\WObj:=wPaper;
    MoveL Offs(pOrigin,121.67,130.97,0.00),v40,z0,tPen\WObj:=wPaper;
    MoveL Offs(pOrigin,120.77,130.37,0.00),v40,z0,tPen\WObj:=wPaper;
    MoveL Offs(pOrigin,118.67,132.47,0.00),v40,z0,tPen\WObj:=wPaper;
    MoveL Offs(pOrigin,118.89,131.86,0.00),v40,z0,tPen\WObj:=wPaper;
    MoveL Offs(pOrigin,119.74,132.71,0.00),v40,z0,tPen\WObj:=wPaper;
    MoveL Offs(pOrigin,118.89,131.86,0.00),v40,z0,tPen\WObj:=wPaper;
    MoveL Offs(pOrigin,118.89,131.16,0.00),v40,z0,tPen\WObj:=wPaper;
    MoveL Offs(pOrigin,120.38,131.16,0.00),v40,fine,tPen\WObj:=wPaper;
    MoveL Offs(pOrigin,120.38,131.16,6.00),v60,z5,tPen\WObj:=wPaper;
    MoveL Offs(pOrigin,119.74,132.22,6.00),vTravel,z5,tPen\WObj:=wPaper;
    MoveL Offs(pOrigin,119.74,132.22,0.00),v60,z0,tPen\WObj:=wPaper;
    MoveL Offs(pOrigin,130.79,132.22,0.00),v40,fine,tPen\WObj:=wPaper;
    MoveL Offs(pOrigin,130.79,132.22,6.00),v60,z5,tPen\WObj:=wPaper;
    MoveL Offs(pOrigin,129.79,133.07,6.00),vTravel,z5,tPen\WObj:=wPaper;
    MoveL Offs(pOrigin,129.79,133.07,0.00),v60,z0,tPen\WObj:=wPaper;
    MoveL Offs(pOrigin,128.44,131.72,0.00),v40,z0,tPen\WObj:=wPaper;
    MoveL Offs(pOrigin,127.51,131.10,0.00),v40,z0,tPen\WObj:=wPaper;
    MoveL Offs(pOrigin,122.70,135.91,0.00),v40,z0,tPen\WObj:=wPaper;
    MoveL Offs(pOrigin,123.56,135.38,0.00),v40,z0,tPen\WObj:=wPaper;
    MoveL Offs(pOrigin,124.62,135.38,0.00),v40,z0,tPen\WObj:=wPaper;
    MoveL Offs(pOrigin,125.05,136.44,0.00),v40,z0,tPen\WObj:=wPaper;
    MoveL Offs(pOrigin,123.78,136.44,0.00),v40,fine,tPen\WObj:=wPaper;
  ENDPROC

  PROC DrawPart41()
    MoveL Offs(pOrigin,123.78,136.44,6.00),v60,z5,tPen\WObj:=wPaper;
    MoveL Offs(pOrigin,123.57,134.41,6.00),vTravel,z5,tPen\WObj:=wPaper;
    MoveL Offs(pOrigin,123.57,134.41,0.00),v60,z0,tPen\WObj:=wPaper;
    MoveL Offs(pOrigin,123.57,132.92,0.00),v40,z0,tPen\WObj:=wPaper;
    MoveL Offs(pOrigin,124.25,132.01,0.00),v40,z0,tPen\WObj:=wPaper;
    MoveL Offs(pOrigin,126.05,133.81,0.00),v40,z0,tPen\WObj:=wPaper;
    MoveL Offs(pOrigin,125.69,133.27,0.00),v40,z0,tPen\WObj:=wPaper;
    MoveL Offs(pOrigin,121.86,133.27,0.00),v40,z0,tPen\WObj:=wPaper;
    MoveL Offs(pOrigin,121.36,134.26,0.00),v40,z0,tPen\WObj:=wPaper;
    MoveL Offs(pOrigin,124.21,131.41,0.00),v40,fine,tPen\WObj:=wPaper;
    MoveL Offs(pOrigin,124.21,131.41,6.00),v60,z5,tPen\WObj:=wPaper;
    MoveL Offs(pOrigin,126.94,131.72,6.00),vTravel,z5,tPen\WObj:=wPaper;
    MoveL Offs(pOrigin,126.94,131.72,0.00),v60,z0,tPen\WObj:=wPaper;
    MoveL Offs(pOrigin,128.60,133.37,0.00),v40,z0,tPen\WObj:=wPaper;
    MoveL Offs(pOrigin,129.60,133.49,0.00),v40,z0,tPen\WObj:=wPaper;
    MoveL Offs(pOrigin,133.06,130.03,0.00),v40,z0,tPen\WObj:=wPaper;
    MoveL Offs(pOrigin,133.53,130.84,0.00),v40,z0,tPen\WObj:=wPaper;
    MoveL Offs(pOrigin,134.89,132.19,0.00),v40,z0,tPen\WObj:=wPaper;
    MoveL Offs(pOrigin,134.85,132.72,0.00),v40,z0,tPen\WObj:=wPaper;
    MoveL Offs(pOrigin,138.60,128.97,0.00),v40,z0,tPen\WObj:=wPaper;
    MoveL Offs(pOrigin,138.47,129.81,0.00),v40,z0,tPen\WObj:=wPaper;
    MoveL Offs(pOrigin,139.68,131.01,0.00),v40,z0,tPen\WObj:=wPaper;
    MoveL Offs(pOrigin,140.84,131.21,0.00),v40,z0,tPen\WObj:=wPaper;
    MoveL Offs(pOrigin,144.75,127.30,0.00),v40,fine,tPen\WObj:=wPaper;
    MoveL Offs(pOrigin,144.75,127.30,6.00),v60,z5,tPen\WObj:=wPaper;
    MoveL Offs(pOrigin,143.11,128.47,6.00),vTravel,z5,tPen\WObj:=wPaper;
    MoveL Offs(pOrigin,143.11,128.47,0.00),v60,z0,tPen\WObj:=wPaper;
    MoveL Offs(pOrigin,144.31,129.67,0.00),v40,fine,tPen\WObj:=wPaper;
    MoveL Offs(pOrigin,144.31,129.67,6.00),v60,z5,tPen\WObj:=wPaper;
    MoveL Offs(pOrigin,147.17,131.03,6.00),vTravel,z5,tPen\WObj:=wPaper;
    MoveL Offs(pOrigin,147.17,131.03,0.00),v60,z0,tPen\WObj:=wPaper;
    MoveL Offs(pOrigin,147.92,131.78,0.00),v40,z0,tPen\WObj:=wPaper;
    MoveL Offs(pOrigin,148.93,132.08,0.00),v40,z0,tPen\WObj:=wPaper;
    MoveL Offs(pOrigin,162.45,118.56,0.00),v40,z0,tPen\WObj:=wPaper;
    MoveL Offs(pOrigin,161.60,118.49,0.00),v40,z0,tPen\WObj:=wPaper;
    MoveL Offs(pOrigin,160.11,118.49,0.00),v40,fine,tPen\WObj:=wPaper;
    MoveL Offs(pOrigin,160.11,118.49,6.00),v60,z5,tPen\WObj:=wPaper;
    MoveL Offs(pOrigin,159.01,117.52,6.00),vTravel,z5,tPen\WObj:=wPaper;
    MoveL Offs(pOrigin,159.01,117.52,0.00),v60,z0,tPen\WObj:=wPaper;
    MoveL Offs(pOrigin,167.73,108.80,0.00),v40,z0,tPen\WObj:=wPaper;
    MoveL Offs(pOrigin,167.32,109.37,0.00),v40,z0,tPen\WObj:=wPaper;
    MoveL Offs(pOrigin,160.56,102.61,0.00),v40,z0,tPen\WObj:=wPaper;
    MoveL Offs(pOrigin,160.75,102.96,0.00),v40,z0,tPen\WObj:=wPaper;
    MoveL Offs(pOrigin,160.54,103.39,0.00),v40,z0,tPen\WObj:=wPaper;
    MoveL Offs(pOrigin,160.75,102.96,0.00),v40,z0,tPen\WObj:=wPaper;
    MoveL Offs(pOrigin,160.96,102.65,0.00),v40,z0,tPen\WObj:=wPaper;
    MoveL Offs(pOrigin,164.15,102.65,0.00),v40,z0,tPen\WObj:=wPaper;
    MoveL Offs(pOrigin,163.69,101.90,0.00),v40,z0,tPen\WObj:=wPaper;
    MoveL Offs(pOrigin,163.69,105.72,0.00),v40,z0,tPen\WObj:=wPaper;
    MoveL Offs(pOrigin,164.15,106.36,0.00),v40,z0,tPen\WObj:=wPaper;
    MoveL Offs(pOrigin,163.73,107.43,0.00),v40,z0,tPen\WObj:=wPaper;
    MoveL Offs(pOrigin,164.50,109.97,0.00),v40,z0,tPen\WObj:=wPaper;
    MoveL Offs(pOrigin,165.71,112.31,0.00),v40,z0,tPen\WObj:=wPaper;
    MoveL Offs(pOrigin,165.85,113.59,0.00),v40,z0,tPen\WObj:=wPaper;
    MoveL Offs(pOrigin,166.28,112.81,0.00),v40,z0,tPen\WObj:=wPaper;
    MoveL Offs(pOrigin,161.17,107.71,0.00),v40,z0,tPen\WObj:=wPaper;
    MoveL Offs(pOrigin,161.60,107.93,0.00),v40,z0,tPen\WObj:=wPaper;
    MoveL Offs(pOrigin,164.36,107.93,0.00),v40,z0,tPen\WObj:=wPaper;
    MoveL Offs(pOrigin,165.00,107.21,0.00),v40,z0,tPen\WObj:=wPaper;
    MoveL Offs(pOrigin,165.21,107.64,0.00),v40,z0,tPen\WObj:=wPaper;
    MoveL Offs(pOrigin,165.00,107.21,0.00),v40,z0,tPen\WObj:=wPaper;
    MoveL Offs(pOrigin,164.79,106.87,0.00),v40,z0,tPen\WObj:=wPaper;
    MoveL Offs(pOrigin,161.81,106.87,0.00),v40,z0,tPen\WObj:=wPaper;
    MoveL Offs(pOrigin,161.81,105.82,0.00),v40,z0,tPen\WObj:=wPaper;
    MoveL Offs(pOrigin,164.58,105.82,0.00),v40,z0,tPen\WObj:=wPaper;
    MoveL Offs(pOrigin,165.21,105.77,0.00),v40,z0,tPen\WObj:=wPaper;
    MoveL Offs(pOrigin,161.16,101.71,0.00),v40,z0,tPen\WObj:=wPaper;
    MoveL Offs(pOrigin,161.60,101.59,0.00),v40,z0,tPen\WObj:=wPaper;
    MoveL Offs(pOrigin,164.15,101.59,0.00),v40,z0,tPen\WObj:=wPaper;
    MoveL Offs(pOrigin,164.15,100.54,0.00),v40,z0,tPen\WObj:=wPaper;
    MoveL Offs(pOrigin,161.81,100.54,0.00),v40,z0,tPen\WObj:=wPaper;
    MoveL Offs(pOrigin,162.02,100.41,0.00),v40,z0,tPen\WObj:=wPaper;
    MoveL Offs(pOrigin,161.67,102.11,0.00),v40,z0,tPen\WObj:=wPaper;
    MoveL Offs(pOrigin,160.11,103.60,0.00),v40,fine,tPen\WObj:=wPaper;
    MoveL Offs(pOrigin,160.11,103.60,6.00),v60,z5,tPen\WObj:=wPaper;
    MoveL Offs(pOrigin,161.58,104.24,6.00),vTravel,z5,tPen\WObj:=wPaper;
    MoveL Offs(pOrigin,161.58,104.24,0.00),v60,z0,tPen\WObj:=wPaper;
    MoveL Offs(pOrigin,161.58,102.75,0.00),v40,z0,tPen\WObj:=wPaper;
    MoveL Offs(pOrigin,161.60,101.90,0.00),v40,z0,tPen\WObj:=wPaper;
    MoveL Offs(pOrigin,161.39,102.32,0.00),v40,z0,tPen\WObj:=wPaper;
    MoveL Offs(pOrigin,161.60,101.90,0.00),v40,fine,tPen\WObj:=wPaper;
    MoveL Offs(pOrigin,161.60,101.90,6.00),v60,z5,tPen\WObj:=wPaper;
    MoveL Offs(pOrigin,160.41,101.19,6.00),vTravel,z5,tPen\WObj:=wPaper;
    MoveL Offs(pOrigin,160.41,101.19,0.00),v60,z0,tPen\WObj:=wPaper;
    MoveL Offs(pOrigin,187.01,74.59,0.00),v40,z0,tPen\WObj:=wPaper;
    MoveL Offs(pOrigin,187.14,75.43,0.00),v40,z0,tPen\WObj:=wPaper;
    MoveL Offs(pOrigin,191.50,79.79,0.00),v40,z0,tPen\WObj:=wPaper;
    MoveL Offs(pOrigin,190.92,79.42,0.00),v40,z0,tPen\WObj:=wPaper;
    MoveL Offs(pOrigin,188.38,79.42,0.00),v40,z0,tPen\WObj:=wPaper;
    MoveL Offs(pOrigin,188.38,79.80,0.00),v40,z0,tPen\WObj:=wPaper;
    MoveL Offs(pOrigin,186.75,80.01,0.00),v40,z0,tPen\WObj:=wPaper;
    MoveL Offs(pOrigin,186.68,81.71,0.00),v40,z0,tPen\WObj:=wPaper;
    MoveL Offs(pOrigin,186.68,81.71,0.00),v40,z0,tPen\WObj:=wPaper;
    MoveL Offs(pOrigin,184.12,84.05,0.00),v40,z0,tPen\WObj:=wPaper;
    MoveL Offs(pOrigin,184.34,83.64,0.00),v40,z0,tPen\WObj:=wPaper;
    MoveL Offs(pOrigin,187.52,83.64,0.00),v40,z0,tPen\WObj:=wPaper;
    MoveL Offs(pOrigin,187.10,84.26,0.00),v40,z0,tPen\WObj:=wPaper;
    MoveL Offs(pOrigin,186.25,85.11,0.00),v40,z0,tPen\WObj:=wPaper;
    MoveL Offs(pOrigin,187.10,84.26,0.00),v40,z0,tPen\WObj:=wPaper;
    MoveL Offs(pOrigin,187.32,84.57,0.00),v40,z0,tPen\WObj:=wPaper;
    MoveL Offs(pOrigin,184.76,82.01,0.00),v40,z0,tPen\WObj:=wPaper;
    MoveL Offs(pOrigin,184.02,82.76,0.00),v40,z0,tPen\WObj:=wPaper;
    MoveL Offs(pOrigin,186.42,85.16,0.00),v40,z0,tPen\WObj:=wPaper;
    MoveL Offs(pOrigin,186.25,84.70,0.00),v40,z0,tPen\WObj:=wPaper;
    MoveL Offs(pOrigin,183.06,84.70,0.00),v40,z0,tPen\WObj:=wPaper;
    MoveL Offs(pOrigin,183.70,84.26,0.00),v40,z0,tPen\WObj:=wPaper;
    MoveL Offs(pOrigin,179.02,88.51,0.00),v40,z0,tPen\WObj:=wPaper;
    MoveL Offs(pOrigin,171.16,94.89,0.00),v40,z0,tPen\WObj:=wPaper;
    MoveL Offs(pOrigin,170.10,95.53,0.00),v40,z0,tPen\WObj:=wPaper;
    MoveL Offs(pOrigin,168.82,95.53,0.00),v40,z0,tPen\WObj:=wPaper;
    MoveL Offs(pOrigin,168.82,95.53,0.00),v40,z0,tPen\WObj:=wPaper;
    MoveL Offs(pOrigin,168.05,94.25,0.00),v40,z0,tPen\WObj:=wPaper;
    MoveL Offs(pOrigin,168.05,93.61,0.00),v40,z0,tPen\WObj:=wPaper;
    MoveL Offs(pOrigin,169.46,92.76,0.00),v40,z0,tPen\WObj:=wPaper;
    MoveL Offs(pOrigin,170.38,91.06,0.00),v40,z0,tPen\WObj:=wPaper;
    MoveL Offs(pOrigin,175.20,86.81,0.00),v40,z0,tPen\WObj:=wPaper;
    MoveL Offs(pOrigin,175.64,87.83,0.00),v40,z0,tPen\WObj:=wPaper;
    MoveL Offs(pOrigin,172.79,84.97,0.00),v40,z0,tPen\WObj:=wPaper;
    MoveL Offs(pOrigin,172.65,85.32,0.00),v40,z0,tPen\WObj:=wPaper;
    MoveL Offs(pOrigin,170.95,87.03,0.00),v40,z0,tPen\WObj:=wPaper;
  ENDPROC

  PROC DrawPart42()
    MoveL Offs(pOrigin,172.65,85.32,0.00),v40,z0,tPen\WObj:=wPaper;
    MoveL Offs(pOrigin,172.44,85.75,0.00),v40,z0,tPen\WObj:=wPaper;
    MoveL Offs(pOrigin,174.56,85.75,0.00),v40,fine,tPen\WObj:=wPaper;
    MoveL Offs(pOrigin,174.56,85.75,6.00),v60,z5,tPen\WObj:=wPaper;
    MoveL Offs(pOrigin,173.71,86.81,6.00),vTravel,z5,tPen\WObj:=wPaper;
    MoveL Offs(pOrigin,173.71,86.81,0.00),v60,z0,tPen\WObj:=wPaper;
    MoveL Offs(pOrigin,171.38,86.81,0.00),v40,z0,tPen\WObj:=wPaper;
    MoveL Offs(pOrigin,171.30,86.46,0.00),v40,z0,tPen\WObj:=wPaper;
    MoveL Offs(pOrigin,174.15,89.32,0.00),v40,z0,tPen\WObj:=wPaper;
    MoveL Offs(pOrigin,174.90,88.57,0.00),v40,z0,tPen\WObj:=wPaper;
    MoveL Offs(pOrigin,172.04,85.72,0.00),v40,fine,tPen\WObj:=wPaper;
    MoveL Offs(pOrigin,172.04,85.72,6.00),v60,z5,tPen\WObj:=wPaper;
    MoveL Offs(pOrigin,173.50,84.70,6.00),vTravel,z5,tPen\WObj:=wPaper;
    MoveL Offs(pOrigin,173.50,84.70,0.00),v60,z0,tPen\WObj:=wPaper;
    MoveL Offs(pOrigin,175.62,84.70,0.00),v40,fine,tPen\WObj:=wPaper;
    MoveL Offs(pOrigin,175.62,84.70,6.00),v60,z5,tPen\WObj:=wPaper;
    MoveL Offs(pOrigin,174.78,83.64,6.00),vTravel,z5,tPen\WObj:=wPaper;
    MoveL Offs(pOrigin,174.78,83.64,0.00),v60,z0,tPen\WObj:=wPaper;
    MoveL Offs(pOrigin,176.90,83.64,0.00),v40,fine,tPen\WObj:=wPaper;
    MoveL Offs(pOrigin,176.90,83.64,6.00),v60,z5,tPen\WObj:=wPaper;
    MoveL Offs(pOrigin,176.05,82.58,6.00),vTravel,z5,tPen\WObj:=wPaper;
    MoveL Offs(pOrigin,176.05,82.58,0.00),v60,z0,tPen\WObj:=wPaper;
    MoveL Offs(pOrigin,178.18,82.58,0.00),v40,fine,tPen\WObj:=wPaper;
    MoveL Offs(pOrigin,178.18,82.58,6.00),v60,z5,tPen\WObj:=wPaper;
    MoveL Offs(pOrigin,176.82,81.54,6.00),vTravel,z5,tPen\WObj:=wPaper;
    MoveL Offs(pOrigin,176.82,81.54,0.00),v60,z0,tPen\WObj:=wPaper;
    MoveL Offs(pOrigin,179.53,84.24,0.00),v40,z0,tPen\WObj:=wPaper;
    MoveL Offs(pOrigin,178.93,85.14,0.00),v40,z0,tPen\WObj:=wPaper;
    MoveL Offs(pOrigin,176.08,82.28,0.00),v40,z0,tPen\WObj:=wPaper;
    MoveL Offs(pOrigin,175.18,82.88,0.00),v40,z0,tPen\WObj:=wPaper;
    MoveL Offs(pOrigin,178.03,85.74,0.00),v40,z0,tPen\WObj:=wPaper;
    MoveL Offs(pOrigin,177.14,86.33,0.00),v40,z0,tPen\WObj:=wPaper;
    MoveL Offs(pOrigin,174.43,83.63,0.00),v40,z0,tPen\WObj:=wPaper;
    MoveL Offs(pOrigin,174.35,83.84,0.00),v40,z0,tPen\WObj:=wPaper;
    MoveL Offs(pOrigin,173.29,84.90,0.00),v40,z0,tPen\WObj:=wPaper;
    MoveL Offs(pOrigin,174.35,83.84,0.00),v40,z0,tPen\WObj:=wPaper;
    MoveL Offs(pOrigin,173.69,84.37,0.00),v40,z0,tPen\WObj:=wPaper;
    MoveL Offs(pOrigin,176.39,87.08,0.00),v40,fine,tPen\WObj:=wPaper;
    MoveL Offs(pOrigin,176.39,87.08,6.00),v60,z5,tPen\WObj:=wPaper;
    MoveL Offs(pOrigin,177.59,88.28,6.00),vTravel,z5,tPen\WObj:=wPaper;
    MoveL Offs(pOrigin,177.59,88.28,0.00),v60,z0,tPen\WObj:=wPaper;
    MoveL Offs(pOrigin,180.15,90.84,0.00),v40,z0,tPen\WObj:=wPaper;
    MoveL Offs(pOrigin,179.45,90.85,0.00),v40,z0,tPen\WObj:=wPaper;
    MoveL Offs(pOrigin,178.60,91.70,0.00),v40,z0,tPen\WObj:=wPaper;
    MoveL Offs(pOrigin,179.45,90.85,0.00),v40,z0,tPen\WObj:=wPaper;
    MoveL Offs(pOrigin,179.02,91.03,0.00),v40,z0,tPen\WObj:=wPaper;
    MoveL Offs(pOrigin,175.41,91.03,0.00),v40,z0,tPen\WObj:=wPaper;
    MoveL Offs(pOrigin,175.20,90.37,0.00),v40,z0,tPen\WObj:=wPaper;
    MoveL Offs(pOrigin,177.76,92.93,0.00),v40,z0,tPen\WObj:=wPaper;
    MoveL Offs(pOrigin,177.96,92.76,0.00),v40,z0,tPen\WObj:=wPaper;
    MoveL Offs(pOrigin,177.11,92.97,0.00),v40,z0,tPen\WObj:=wPaper;
    MoveL Offs(pOrigin,173.50,95.81,0.00),v40,z0,tPen\WObj:=wPaper;
    MoveL Offs(pOrigin,173.29,96.59,0.00),v40,z0,tPen\WObj:=wPaper;
    MoveL Offs(pOrigin,173.29,96.59,0.00),v40,z0,tPen\WObj:=wPaper;
    MoveL Offs(pOrigin,172.44,96.59,0.00),v40,z0,tPen\WObj:=wPaper;
    MoveL Offs(pOrigin,168.61,97.86,0.00),v40,z0,tPen\WObj:=wPaper;
    MoveL Offs(pOrigin,167.55,97.86,0.00),v40,z0,tPen\WObj:=wPaper;
    MoveL Offs(pOrigin,165.85,96.87,0.00),v40,z0,tPen\WObj:=wPaper;
    MoveL Offs(pOrigin,165.21,96.87,0.00),v40,z0,tPen\WObj:=wPaper;
    MoveL Offs(pOrigin,164.15,100.20,0.00),v40,z0,tPen\WObj:=wPaper;
    MoveL Offs(pOrigin,164.36,104.88,0.00),v40,z0,tPen\WObj:=wPaper;
    MoveL Offs(pOrigin,164.01,105.72,0.00),v40,z0,tPen\WObj:=wPaper;
    MoveL Offs(pOrigin,170.10,114.37,0.00),v40,z0,tPen\WObj:=wPaper;
    MoveL Offs(pOrigin,170.88,114.72,0.00),v40,z0,tPen\WObj:=wPaper;
    MoveL Offs(pOrigin,171.38,115.93,0.00),v40,z0,tPen\WObj:=wPaper;
    MoveL Offs(pOrigin,171.94,116.21,0.00),v40,z0,tPen\WObj:=wPaper;
    MoveL Offs(pOrigin,172.51,117.41,0.00),v40,z0,tPen\WObj:=wPaper;
    MoveL Offs(pOrigin,173.00,117.70,0.00),v40,z0,tPen\WObj:=wPaper;
    MoveL Offs(pOrigin,177.18,124.21,0.00),v40,z0,tPen\WObj:=wPaper;
    MoveL Offs(pOrigin,179.52,128.89,0.00),v40,z0,tPen\WObj:=wPaper;
    MoveL Offs(pOrigin,182.21,136.54,0.00),v40,z0,tPen\WObj:=wPaper;
    MoveL Offs(pOrigin,182.00,137.18,0.00),v40,z0,tPen\WObj:=wPaper;
    MoveL Offs(pOrigin,182.00,137.18,0.00),v40,z0,tPen\WObj:=wPaper;
    MoveL Offs(pOrigin,183.49,144.40,0.00),v40,z0,tPen\WObj:=wPaper;
    MoveL Offs(pOrigin,183.91,151.20,0.00),v40,fine,tPen\WObj:=wPaper;
    MoveL Offs(pOrigin,183.91,151.20,6.00),v60,z5,tPen\WObj:=wPaper;
    MoveL Offs(pOrigin,183.18,148.60,6.00),vTravel,z5,tPen\WObj:=wPaper;
    MoveL Offs(pOrigin,183.18,148.60,0.00),v60,z0,tPen\WObj:=wPaper;
    MoveL Offs(pOrigin,184.23,147.55,0.00),v40,fine,tPen\WObj:=wPaper;
    MoveL Offs(pOrigin,184.23,147.55,6.00),v60,z5,tPen\WObj:=wPaper;
    MoveL Offs(pOrigin,182.89,147.41,6.00),vTravel,z5,tPen\WObj:=wPaper;
    MoveL Offs(pOrigin,182.89,147.41,0.00),v60,z0,tPen\WObj:=wPaper;
    MoveL Offs(pOrigin,184.24,146.05,0.00),v40,fine,tPen\WObj:=wPaper;
    MoveL Offs(pOrigin,184.24,146.05,6.00),v60,z5,tPen\WObj:=wPaper;
    MoveL Offs(pOrigin,182.74,146.06,6.00),vTravel,z5,tPen\WObj:=wPaper;
    MoveL Offs(pOrigin,182.74,146.06,0.00),v60,z0,tPen\WObj:=wPaper;
    MoveL Offs(pOrigin,184.24,144.56,0.00),v40,fine,tPen\WObj:=wPaper;
    MoveL Offs(pOrigin,184.24,144.56,6.00),v60,z5,tPen\WObj:=wPaper;
    MoveL Offs(pOrigin,184.10,143.21,6.00),vTravel,z5,tPen\WObj:=wPaper;
    MoveL Offs(pOrigin,184.10,143.21,0.00),v60,z0,tPen\WObj:=wPaper;
    MoveL Offs(pOrigin,182.45,144.86,0.00),v40,fine,tPen\WObj:=wPaper;
    MoveL Offs(pOrigin,182.45,144.86,6.00),v60,z5,tPen\WObj:=wPaper;
    MoveL Offs(pOrigin,182.30,143.51,6.00),vTravel,z5,tPen\WObj:=wPaper;
    MoveL Offs(pOrigin,182.30,143.51,0.00),v60,z0,tPen\WObj:=wPaper;
    MoveL Offs(pOrigin,184.10,141.71,0.00),v40,z0,tPen\WObj:=wPaper;
    MoveL Offs(pOrigin,183.15,141.63,0.00),v40,z0,tPen\WObj:=wPaper;
    MoveL Offs(pOrigin,182.25,140.73,0.00),v40,z0,tPen\WObj:=wPaper;
    MoveL Offs(pOrigin,181.71,141.12,0.00),v40,z0,tPen\WObj:=wPaper;
    MoveL Offs(pOrigin,183.66,139.16,0.00),v40,z0,tPen\WObj:=wPaper;
    MoveL Offs(pOrigin,182.99,139.98,0.00),v40,z0,tPen\WObj:=wPaper;
    MoveL Offs(pOrigin,181.79,138.78,0.00),v40,z0,tPen\WObj:=wPaper;
    MoveL Offs(pOrigin,181.27,138.57,0.00),v40,z0,tPen\WObj:=wPaper;
    MoveL Offs(pOrigin,183.07,136.77,0.00),v40,z0,tPen\WObj:=wPaper;
    MoveL Offs(pOrigin,182.62,135.72,0.00),v40,z0,tPen\WObj:=wPaper;
    MoveL Offs(pOrigin,180.82,137.53,0.00),v40,z0,tPen\WObj:=wPaper;
    MoveL Offs(pOrigin,181.04,136.53,0.00),v40,z0,tPen\WObj:=wPaper;
    MoveL Offs(pOrigin,182.54,138.03,0.00),v40,z0,tPen\WObj:=wPaper;
    MoveL Offs(pOrigin,183.22,138.12,0.00),v40,z0,tPen\WObj:=wPaper;
    MoveL Offs(pOrigin,181.41,139.92,0.00),v40,fine,tPen\WObj:=wPaper;
    MoveL Offs(pOrigin,181.41,139.92,6.00),v60,z5,tPen\WObj:=wPaper;
    MoveL Offs(pOrigin,182.15,142.16,6.00),vTravel,z5,tPen\WObj:=wPaper;
    MoveL Offs(pOrigin,182.15,142.16,0.00),v60,z0,tPen\WObj:=wPaper;
    MoveL Offs(pOrigin,183.81,140.51,0.00),v40,fine,tPen\WObj:=wPaper;
    MoveL Offs(pOrigin,183.81,140.51,6.00),v60,z5,tPen\WObj:=wPaper;
    MoveL Offs(pOrigin,182.00,137.18,6.00),vTravel,z5,tPen\WObj:=wPaper;
    MoveL Offs(pOrigin,182.00,137.18,0.00),v60,z0,tPen\WObj:=wPaper;
    MoveL Offs(pOrigin,181.43,136.75,0.00),v40,z0,tPen\WObj:=wPaper;
    MoveL Offs(pOrigin,179.95,132.29,0.00),v40,z0,tPen\WObj:=wPaper;
    MoveL Offs(pOrigin,177.47,126.76,0.00),v40,z0,tPen\WObj:=wPaper;
    MoveL Offs(pOrigin,172.01,117.84,0.00),v40,z0,tPen\WObj:=wPaper;
  ENDPROC

  PROC DrawPart43()
    MoveL Offs(pOrigin,172.01,117.84,0.00),v40,z0,tPen\WObj:=wPaper;
    MoveL Offs(pOrigin,170.88,115.93,0.00),v40,z0,tPen\WObj:=wPaper;
    MoveL Offs(pOrigin,170.17,115.43,0.00),v40,z0,tPen\WObj:=wPaper;
    MoveL Offs(pOrigin,169.89,114.44,0.00),v40,fine,tPen\WObj:=wPaper;
    MoveL Offs(pOrigin,169.89,114.44,6.00),v60,z5,tPen\WObj:=wPaper;
    MoveL Offs(pOrigin,168.08,113.12,6.00),vTravel,z5,tPen\WObj:=wPaper;
    MoveL Offs(pOrigin,168.08,113.12,0.00),v60,z0,tPen\WObj:=wPaper;
    MoveL Offs(pOrigin,174.54,119.58,0.00),v40,z0,tPen\WObj:=wPaper;
    MoveL Offs(pOrigin,175.03,119.42,0.00),v40,z0,tPen\WObj:=wPaper;
    MoveL Offs(pOrigin,173.08,121.37,0.00),v40,z0,tPen\WObj:=wPaper;
    MoveL Offs(pOrigin,173.83,122.12,0.00),v40,z0,tPen\WObj:=wPaper;
    MoveL Offs(pOrigin,175.48,120.46,0.00),v40,z0,tPen\WObj:=wPaper;
    MoveL Offs(pOrigin,174.99,120.81,0.00),v40,z0,tPen\WObj:=wPaper;
    MoveL Offs(pOrigin,175.20,121.24,0.00),v40,z0,tPen\WObj:=wPaper;
    MoveL Offs(pOrigin,174.99,120.81,0.00),v40,fine,tPen\WObj:=wPaper;
    MoveL Offs(pOrigin,174.99,120.81,6.00),v60,z5,tPen\WObj:=wPaper;
    MoveL Offs(pOrigin,174.55,122.58,6.00),vTravel,z5,tPen\WObj:=wPaper;
    MoveL Offs(pOrigin,174.55,122.58,0.00),v60,z0,tPen\WObj:=wPaper;
    MoveL Offs(pOrigin,178.61,126.63,0.00),v40,z0,tPen\WObj:=wPaper;
    MoveL Offs(pOrigin,178.76,126.15,0.00),v40,z0,tPen\WObj:=wPaper;
    MoveL Offs(pOrigin,177.11,127.80,0.00),v40,z0,tPen\WObj:=wPaper;
    MoveL Offs(pOrigin,176.36,127.05,0.00),v40,z0,tPen\WObj:=wPaper;
    MoveL Offs(pOrigin,178.46,124.95,0.00),v40,z0,tPen\WObj:=wPaper;
    MoveL Offs(pOrigin,178.02,123.90,0.00),v40,z0,tPen\WObj:=wPaper;
    MoveL Offs(pOrigin,176.06,125.86,0.00),v40,z0,tPen\WObj:=wPaper;
    MoveL Offs(pOrigin,176.66,126.18,0.00),v40,z0,tPen\WObj:=wPaper;
    MoveL Offs(pOrigin,179.97,129.48,0.00),v40,z0,tPen\WObj:=wPaper;
    MoveL Offs(pOrigin,180.25,129.14,0.00),v40,z0,tPen\WObj:=wPaper;
    MoveL Offs(pOrigin,178.44,130.94,0.00),v40,z0,tPen\WObj:=wPaper;
    MoveL Offs(pOrigin,178.89,131.99,0.00),v40,z0,tPen\WObj:=wPaper;
    MoveL Offs(pOrigin,180.69,130.19,0.00),v40,z0,tPen\WObj:=wPaper;
    MoveL Offs(pOrigin,181.14,131.23,0.00),v40,z0,tPen\WObj:=wPaper;
    MoveL Offs(pOrigin,179.34,133.04,0.00),v40,z0,tPen\WObj:=wPaper;
    MoveL Offs(pOrigin,179.37,131.88,0.00),v40,z0,tPen\WObj:=wPaper;
    MoveL Offs(pOrigin,181.63,134.13,0.00),v40,z0,tPen\WObj:=wPaper;
    MoveL Offs(pOrigin,182.33,134.52,0.00),v40,z0,tPen\WObj:=wPaper;
    MoveL Offs(pOrigin,180.37,136.48,0.00),v40,fine,tPen\WObj:=wPaper;
    MoveL Offs(pOrigin,180.37,136.48,6.00),v60,z5,tPen\WObj:=wPaper;
    MoveL Offs(pOrigin,180.08,135.28,6.00),vTravel,z5,tPen\WObj:=wPaper;
    MoveL Offs(pOrigin,180.08,135.28,0.00),v60,z0,tPen\WObj:=wPaper;
    MoveL Offs(pOrigin,182.03,133.33,0.00),v40,z0,tPen\WObj:=wPaper;
    MoveL Offs(pOrigin,181.59,132.28,0.00),v40,z0,tPen\WObj:=wPaper;
    MoveL Offs(pOrigin,179.63,134.23,0.00),v40,z0,tPen\WObj:=wPaper;
    MoveL Offs(pOrigin,180.13,134.13,0.00),v40,z0,tPen\WObj:=wPaper;
    MoveL Offs(pOrigin,182.08,136.08,0.00),v40,fine,tPen\WObj:=wPaper;
    MoveL Offs(pOrigin,182.08,136.08,6.00),v60,z5,tPen\WObj:=wPaper;
    MoveL Offs(pOrigin,181.02,132.03,6.00),vTravel,z5,tPen\WObj:=wPaper;
    MoveL Offs(pOrigin,181.02,132.03,0.00),v60,z0,tPen\WObj:=wPaper;
    MoveL Offs(pOrigin,178.17,129.18,0.00),v40,z0,tPen\WObj:=wPaper;
    MoveL Offs(pOrigin,178.39,129.10,0.00),v40,z0,tPen\WObj:=wPaper;
    MoveL Offs(pOrigin,178.60,129.52,0.00),v40,z0,tPen\WObj:=wPaper;
    MoveL Offs(pOrigin,178.39,129.10,0.00),v40,z0,tPen\WObj:=wPaper;
    MoveL Offs(pOrigin,177.55,128.85,0.00),v40,z0,tPen\WObj:=wPaper;
    MoveL Offs(pOrigin,179.50,126.89,0.00),v40,z0,tPen\WObj:=wPaper;
    MoveL Offs(pOrigin,179.95,127.94,0.00),v40,z0,tPen\WObj:=wPaper;
    MoveL Offs(pOrigin,178.00,129.89,0.00),v40,fine,tPen\WObj:=wPaper;
    MoveL Offs(pOrigin,178.00,129.89,6.00),v60,z5,tPen\WObj:=wPaper;
    MoveL Offs(pOrigin,174.40,132.00,6.00),vTravel,z5,tPen\WObj:=wPaper;
    MoveL Offs(pOrigin,174.40,132.00,0.00),v60,z0,tPen\WObj:=wPaper;
    MoveL Offs(pOrigin,173.04,133.35,0.00),v40,z0,tPen\WObj:=wPaper;
    MoveL Offs(pOrigin,173.93,133.35,0.00),v40,z0,tPen\WObj:=wPaper;
    MoveL Offs(pOrigin,174.14,133.77,0.00),v40,z0,tPen\WObj:=wPaper;
    MoveL Offs(pOrigin,173.93,133.35,0.00),v40,z0,tPen\WObj:=wPaper;
    MoveL Offs(pOrigin,174.84,133.05,0.00),v40,z0,tPen\WObj:=wPaper;
    MoveL Offs(pOrigin,173.49,134.40,0.00),v40,z0,tPen\WObj:=wPaper;
    MoveL Offs(pOrigin,173.94,135.45,0.00),v40,z0,tPen\WObj:=wPaper;
    MoveL Offs(pOrigin,175.44,133.95,0.00),v40,z0,tPen\WObj:=wPaper;
    MoveL Offs(pOrigin,175.88,134.99,0.00),v40,z0,tPen\WObj:=wPaper;
    MoveL Offs(pOrigin,174.23,136.65,0.00),v40,z0,tPen\WObj:=wPaper;
    MoveL Offs(pOrigin,174.59,136.06,0.00),v40,z0,tPen\WObj:=wPaper;
    MoveL Offs(pOrigin,176.40,137.86,0.00),v40,z0,tPen\WObj:=wPaper;
    MoveL Offs(pOrigin,176.78,137.09,0.00),v40,z0,tPen\WObj:=wPaper;
    MoveL Offs(pOrigin,174.97,138.89,0.00),v40,z0,tPen\WObj:=wPaper;
    MoveL Offs(pOrigin,175.20,138.16,0.00),v40,z0,tPen\WObj:=wPaper;
    MoveL Offs(pOrigin,177.30,140.26,0.00),v40,z0,tPen\WObj:=wPaper;
    MoveL Offs(pOrigin,177.97,140.38,0.00),v40,z0,tPen\WObj:=wPaper;
    MoveL Offs(pOrigin,176.16,142.18,0.00),v40,z0,tPen\WObj:=wPaper;
    MoveL Offs(pOrigin,176.71,142.66,0.00),v40,z0,tPen\WObj:=wPaper;
    MoveL Offs(pOrigin,178.51,144.46,0.00),v40,z0,tPen\WObj:=wPaper;
    MoveL Offs(pOrigin,179.00,143.82,0.00),v40,z0,tPen\WObj:=wPaper;
    MoveL Offs(pOrigin,177.05,145.78,0.00),v40,z0,tPen\WObj:=wPaper;
    MoveL Offs(pOrigin,177.62,146.55,0.00),v40,z0,tPen\WObj:=wPaper;
    MoveL Offs(pOrigin,179.12,148.06,0.00),v40,z0,tPen\WObj:=wPaper;
    MoveL Offs(pOrigin,179.89,147.41,0.00),v40,z0,tPen\WObj:=wPaper;
    MoveL Offs(pOrigin,177.64,149.67,0.00),v40,z0,tPen\WObj:=wPaper;
    MoveL Offs(pOrigin,178.23,150.15,0.00),v40,z0,tPen\WObj:=wPaper;
    MoveL Offs(pOrigin,179.58,151.50,0.00),v40,z0,tPen\WObj:=wPaper;
    MoveL Offs(pOrigin,180.18,151.61,0.00),v40,z0,tPen\WObj:=wPaper;
    MoveL Offs(pOrigin,177.77,154.01,0.00),v40,z0,tPen\WObj:=wPaper;
    MoveL Offs(pOrigin,178.54,153.45,0.00),v40,z0,tPen\WObj:=wPaper;
    MoveL Offs(pOrigin,179.89,154.80,0.00),v40,z0,tPen\WObj:=wPaper;
    MoveL Offs(pOrigin,180.47,154.30,0.00),v40,z0,tPen\WObj:=wPaper;
    MoveL Offs(pOrigin,178.06,156.71,0.00),v40,z0,tPen\WObj:=wPaper;
    MoveL Offs(pOrigin,178.55,156.44,0.00),v40,z0,tPen\WObj:=wPaper;
    MoveL Offs(pOrigin,179.90,157.80,0.00),v40,z0,tPen\WObj:=wPaper;
    MoveL Offs(pOrigin,180.46,157.30,0.00),v40,z0,tPen\WObj:=wPaper;
    MoveL Offs(pOrigin,177.76,160.00,0.00),v40,z0,tPen\WObj:=wPaper;
    MoveL Offs(pOrigin,178.26,160.64,0.00),v40,z0,tPen\WObj:=wPaper;
    MoveL Offs(pOrigin,179.17,161.54,0.00),v40,z0,tPen\WObj:=wPaper;
    MoveL Offs(pOrigin,179.24,161.19,0.00),v40,z0,tPen\WObj:=wPaper;
    MoveL Offs(pOrigin,179.45,159.70,0.00),v40,z0,tPen\WObj:=wPaper;
    MoveL Offs(pOrigin,179.24,159.27,0.00),v40,z0,tPen\WObj:=wPaper;
    MoveL Offs(pOrigin,179.24,159.27,0.00),v40,z0,tPen\WObj:=wPaper;
    MoveL Offs(pOrigin,179.66,158.64,0.00),v40,z0,tPen\WObj:=wPaper;
    MoveL Offs(pOrigin,179.66,152.05,0.00),v40,z0,tPen\WObj:=wPaper;
    MoveL Offs(pOrigin,178.60,145.25,0.00),v40,z0,tPen\WObj:=wPaper;
    MoveL Offs(pOrigin,177.54,141.85,0.00),v40,z0,tPen\WObj:=wPaper;
    MoveL Offs(pOrigin,177.54,141.85,0.00),v40,z0,tPen\WObj:=wPaper;
    MoveL Offs(pOrigin,176.90,142.27,0.00),v40,z0,tPen\WObj:=wPaper;
    MoveL Offs(pOrigin,178.60,150.35,0.00),v40,z0,tPen\WObj:=wPaper;
    MoveL Offs(pOrigin,178.81,158.85,0.00),v40,z0,tPen\WObj:=wPaper;
    MoveL Offs(pOrigin,179.24,159.27,0.00),v40,z0,tPen\WObj:=wPaper;
    MoveL Offs(pOrigin,178.81,159.27,0.00),v40,z0,tPen\WObj:=wPaper;
    MoveL Offs(pOrigin,178.60,161.19,0.00),v40,z0,tPen\WObj:=wPaper;
    MoveL Offs(pOrigin,178.60,161.19,0.00),v40,z0,tPen\WObj:=wPaper;
    MoveL Offs(pOrigin,178.39,162.46,0.00),v40,z0,tPen\WObj:=wPaper;
    MoveL Offs(pOrigin,178.39,162.46,0.00),v40,z0,tPen\WObj:=wPaper;
    MoveL Offs(pOrigin,179.02,162.68,0.00),v40,z0,tPen\WObj:=wPaper;
    MoveL Offs(pOrigin,179.02,163.10,0.00),v40,z0,tPen\WObj:=wPaper;
    MoveL Offs(pOrigin,178.39,163.52,0.00),v40,z0,tPen\WObj:=wPaper;
  ENDPROC

  PROC DrawPart44()
    MoveL Offs(pOrigin,179.02,162.89,0.00),v40,z0,tPen\WObj:=wPaper;
    MoveL Offs(pOrigin,178.27,162.13,0.00),v40,z0,tPen\WObj:=wPaper;
    MoveL Offs(pOrigin,178.39,162.46,0.00),v40,z0,tPen\WObj:=wPaper;
    MoveL Offs(pOrigin,178.32,163.95,0.00),v40,z0,tPen\WObj:=wPaper;
    MoveL Offs(pOrigin,177.40,167.35,0.00),v40,z0,tPen\WObj:=wPaper;
    MoveL Offs(pOrigin,176.12,170.11,0.00),v40,z0,tPen\WObj:=wPaper;
    MoveL Offs(pOrigin,173.71,173.51,0.00),v40,z0,tPen\WObj:=wPaper;
    MoveL Offs(pOrigin,174.12,172.60,0.00),v40,z0,tPen\WObj:=wPaper;
    MoveL Offs(pOrigin,177.28,169.44,0.00),v40,fine,tPen\WObj:=wPaper;
    MoveL Offs(pOrigin,177.28,169.44,6.00),v60,z5,tPen\WObj:=wPaper;
    MoveL Offs(pOrigin,175.93,167.80,6.00),vTravel,z5,tPen\WObj:=wPaper;
    MoveL Offs(pOrigin,175.93,167.80,0.00),v60,z0,tPen\WObj:=wPaper;
    MoveL Offs(pOrigin,179.09,164.64,0.00),v40,z0,tPen\WObj:=wPaper;
    MoveL Offs(pOrigin,178.43,165.28,0.00),v40,z0,tPen\WObj:=wPaper;
    MoveL Offs(pOrigin,177.68,164.53,0.00),v40,z0,tPen\WObj:=wPaper;
    MoveL Offs(pOrigin,177.15,163.60,0.00),v40,z0,tPen\WObj:=wPaper;
    MoveL Offs(pOrigin,180.00,160.75,0.00),v40,z0,tPen\WObj:=wPaper;
    MoveL Offs(pOrigin,179.46,160.34,0.00),v40,z0,tPen\WObj:=wPaper;
    MoveL Offs(pOrigin,178.56,159.44,0.00),v40,z0,tPen\WObj:=wPaper;
    MoveL Offs(pOrigin,179.61,158.99,0.00),v40,z0,tPen\WObj:=wPaper;
    MoveL Offs(pOrigin,178.56,157.94,0.00),v40,z0,tPen\WObj:=wPaper;
    MoveL Offs(pOrigin,177.76,158.51,0.00),v40,z0,tPen\WObj:=wPaper;
    MoveL Offs(pOrigin,180.46,155.80,0.00),v40,z0,tPen\WObj:=wPaper;
    MoveL Offs(pOrigin,179.90,156.30,0.00),v40,z0,tPen\WObj:=wPaper;
    MoveL Offs(pOrigin,178.55,154.95,0.00),v40,z0,tPen\WObj:=wPaper;
    MoveL Offs(pOrigin,177.92,155.36,0.00),v40,z0,tPen\WObj:=wPaper;
    MoveL Offs(pOrigin,180.47,152.81,0.00),v40,z0,tPen\WObj:=wPaper;
    MoveL Offs(pOrigin,179.89,153.30,0.00),v40,z0,tPen\WObj:=wPaper;
    MoveL Offs(pOrigin,178.24,151.65,0.00),v40,z0,tPen\WObj:=wPaper;
    MoveL Offs(pOrigin,177.63,151.17,0.00),v40,z0,tPen\WObj:=wPaper;
    MoveL Offs(pOrigin,180.04,148.76,0.00),v40,fine,tPen\WObj:=wPaper;
    MoveL Offs(pOrigin,180.04,148.76,6.00),v60,z5,tPen\WObj:=wPaper;
    MoveL Offs(pOrigin,179.58,150.00,6.00),vTravel,z5,tPen\WObj:=wPaper;
    MoveL Offs(pOrigin,179.58,150.00,0.00),v60,z0,tPen\WObj:=wPaper;
    MoveL Offs(pOrigin,177.78,148.20,0.00),v40,z0,tPen\WObj:=wPaper;
    MoveL Offs(pOrigin,177.49,148.32,0.00),v40,z0,tPen\WObj:=wPaper;
    MoveL Offs(pOrigin,179.60,146.22,0.00),v40,z0,tPen\WObj:=wPaper;
    MoveL Offs(pOrigin,178.97,146.41,0.00),v40,z0,tPen\WObj:=wPaper;
    MoveL Offs(pOrigin,177.17,144.60,0.00),v40,z0,tPen\WObj:=wPaper;
    MoveL Offs(pOrigin,176.60,144.73,0.00),v40,z0,tPen\WObj:=wPaper;
    MoveL Offs(pOrigin,178.56,142.78,0.00),v40,z0,tPen\WObj:=wPaper;
    MoveL Offs(pOrigin,177.91,142.36,0.00),v40,z0,tPen\WObj:=wPaper;
    MoveL Offs(pOrigin,176.11,140.56,0.00),v40,z0,tPen\WObj:=wPaper;
    MoveL Offs(pOrigin,175.72,141.14,0.00),v40,z0,tPen\WObj:=wPaper;
    MoveL Offs(pOrigin,177.67,139.18,0.00),v40,z0,tPen\WObj:=wPaper;
    MoveL Offs(pOrigin,177.22,138.14,0.00),v40,z0,tPen\WObj:=wPaper;
    MoveL Offs(pOrigin,175.27,140.09,0.00),v40,fine,tPen\WObj:=wPaper;
    MoveL Offs(pOrigin,175.27,140.09,6.00),v60,z5,tPen\WObj:=wPaper;
    MoveL Offs(pOrigin,176.05,138.88,6.00),vTravel,z5,tPen\WObj:=wPaper;
    MoveL Offs(pOrigin,176.05,138.88,0.00),v60,z0,tPen\WObj:=wPaper;
    MoveL Offs(pOrigin,176.90,141.85,0.00),v40,z0,tPen\WObj:=wPaper;
    MoveL Offs(pOrigin,177.54,141.85,0.00),v40,z0,tPen\WObj:=wPaper;
    MoveL Offs(pOrigin,176.83,139.30,0.00),v40,z0,tPen\WObj:=wPaper;
    MoveL Offs(pOrigin,176.05,138.88,0.00),v40,z0,tPen\WObj:=wPaper;
    MoveL Offs(pOrigin,176.05,138.88,0.00),v40,z0,tPen\WObj:=wPaper;
    MoveL Offs(pOrigin,174.42,133.99,0.00),v40,z0,tPen\WObj:=wPaper;
    MoveL Offs(pOrigin,171.16,127.40,0.00),v40,fine,tPen\WObj:=wPaper;
    MoveL Offs(pOrigin,171.16,127.40,6.00),v60,z5,tPen\WObj:=wPaper;
    MoveL Offs(pOrigin,172.61,129.31,6.00),vTravel,z5,tPen\WObj:=wPaper;
    MoveL Offs(pOrigin,172.61,129.31,0.00),v60,z0,tPen\WObj:=wPaper;
    MoveL Offs(pOrigin,171.70,130.21,0.00),v40,z0,tPen\WObj:=wPaper;
    MoveL Offs(pOrigin,172.15,131.26,0.00),v40,z0,tPen\WObj:=wPaper;
    MoveL Offs(pOrigin,173.35,130.06,0.00),v40,z0,tPen\WObj:=wPaper;
    MoveL Offs(pOrigin,173.80,131.11,0.00),v40,z0,tPen\WObj:=wPaper;
    MoveL Offs(pOrigin,172.60,132.31,0.00),v40,fine,tPen\WObj:=wPaper;
    MoveL Offs(pOrigin,172.60,132.31,6.00),v60,z5,tPen\WObj:=wPaper;
    MoveL Offs(pOrigin,176.33,136.04,6.00),vTravel,z5,tPen\WObj:=wPaper;
    MoveL Offs(pOrigin,176.33,136.04,0.00),v60,z0,tPen\WObj:=wPaper;
    MoveL Offs(pOrigin,174.68,137.69,0.00),v40,fine,tPen\WObj:=wPaper;
    MoveL Offs(pOrigin,174.68,137.69,6.00),v60,z5,tPen\WObj:=wPaper;
    MoveL Offs(pOrigin,178.41,141.43,6.00),vTravel,z5,tPen\WObj:=wPaper;
    MoveL Offs(pOrigin,178.41,141.43,0.00),v60,z0,tPen\WObj:=wPaper;
    MoveL Offs(pOrigin,176.31,143.53,0.00),v40,fine,tPen\WObj:=wPaper;
    MoveL Offs(pOrigin,176.31,143.53,6.00),v60,z5,tPen\WObj:=wPaper;
    MoveL Offs(pOrigin,179.15,145.17,6.00),vTravel,z5,tPen\WObj:=wPaper;
    MoveL Offs(pOrigin,179.15,145.17,0.00),v60,z0,tPen\WObj:=wPaper;
    MoveL Offs(pOrigin,177.20,147.12,0.00),v40,fine,tPen\WObj:=wPaper;
    MoveL Offs(pOrigin,177.20,147.12,6.00),v60,z5,tPen\WObj:=wPaper;
    MoveL Offs(pOrigin,180.18,150.11,6.00),vTravel,z5,tPen\WObj:=wPaper;
    MoveL Offs(pOrigin,180.18,150.11,0.00),v60,z0,tPen\WObj:=wPaper;
    MoveL Offs(pOrigin,177.78,152.51,0.00),v40,fine,tPen\WObj:=wPaper;
    MoveL Offs(pOrigin,177.78,152.51,6.00),v60,z5,tPen\WObj:=wPaper;
    MoveL Offs(pOrigin,180.15,159.10,6.00),vTravel,z5,tPen\WObj:=wPaper;
    MoveL Offs(pOrigin,180.15,159.10,0.00),v60,z0,tPen\WObj:=wPaper;
    MoveL Offs(pOrigin,177.60,161.65,0.00),v40,z0,tPen\WObj:=wPaper;
    MoveL Offs(pOrigin,178.60,161.19,0.00),v40,z0,tPen\WObj:=wPaper;
    MoveL Offs(pOrigin,179.24,161.40,0.00),v40,z0,tPen\WObj:=wPaper;
    MoveL Offs(pOrigin,179.02,162.46,0.00),v40,z0,tPen\WObj:=wPaper;
    MoveL Offs(pOrigin,179.85,162.39,0.00),v40,z0,tPen\WObj:=wPaper;
    MoveL Offs(pOrigin,176.54,165.70,0.00),v40,fine,tPen\WObj:=wPaper;
    MoveL Offs(pOrigin,176.54,165.70,6.00),v60,z5,tPen\WObj:=wPaper;
    MoveL Offs(pOrigin,178.48,166.74,6.00),vTravel,z5,tPen\WObj:=wPaper;
    MoveL Offs(pOrigin,178.48,166.74,0.00),v60,z0,tPen\WObj:=wPaper;
    MoveL Offs(pOrigin,174.88,170.35,0.00),v40,fine,tPen\WObj:=wPaper;
    MoveL Offs(pOrigin,174.88,170.35,6.00),v60,z5,tPen\WObj:=wPaper;
    MoveL Offs(pOrigin,187.61,171.06,6.00),vTravel,z5,tPen\WObj:=wPaper;
    MoveL Offs(pOrigin,187.61,171.06,0.00),v60,z0,tPen\WObj:=wPaper;
    MoveL Offs(pOrigin,189.86,168.81,0.00),v40,fine,tPen\WObj:=wPaper;
    MoveL Offs(pOrigin,189.86,168.81,6.00),v60,z5,tPen\WObj:=wPaper;
    MoveL Offs(pOrigin,189.87,167.31,6.00),vTravel,z5,tPen\WObj:=wPaper;
    MoveL Offs(pOrigin,189.87,167.31,0.00),v60,z0,tPen\WObj:=wPaper;
    MoveL Offs(pOrigin,187.61,169.56,0.00),v40,fine,tPen\WObj:=wPaper;
    MoveL Offs(pOrigin,187.61,169.56,6.00),v60,z5,tPen\WObj:=wPaper;
    MoveL Offs(pOrigin,187.92,167.76,6.00),vTravel,z5,tPen\WObj:=wPaper;
    MoveL Offs(pOrigin,187.92,167.76,0.00),v60,z0,tPen\WObj:=wPaper;
    MoveL Offs(pOrigin,189.87,165.81,0.00),v40,fine,tPen\WObj:=wPaper;
    MoveL Offs(pOrigin,189.87,165.81,6.00),v60,z5,tPen\WObj:=wPaper;
    MoveL Offs(pOrigin,190.03,164.16,6.00),vTravel,z5,tPen\WObj:=wPaper;
    MoveL Offs(pOrigin,190.03,164.16,0.00),v60,z0,tPen\WObj:=wPaper;
    MoveL Offs(pOrigin,188.07,166.11,0.00),v40,fine,tPen\WObj:=wPaper;
    MoveL Offs(pOrigin,188.07,166.11,6.00),v60,z5,tPen\WObj:=wPaper;
    MoveL Offs(pOrigin,188.38,164.32,6.00),vTravel,z5,tPen\WObj:=wPaper;
    MoveL Offs(pOrigin,188.38,164.32,0.00),v60,z0,tPen\WObj:=wPaper;
    MoveL Offs(pOrigin,189.88,162.81,0.00),v40,fine,tPen\WObj:=wPaper;
    MoveL Offs(pOrigin,189.88,162.81,6.00),v60,z5,tPen\WObj:=wPaper;
    MoveL Offs(pOrigin,189.44,160.12,6.00),vTravel,z5,tPen\WObj:=wPaper;
    MoveL Offs(pOrigin,189.44,160.12,0.00),v60,z0,tPen\WObj:=wPaper;
    MoveL Offs(pOrigin,189.65,161.40,0.00),v40,z0,tPen\WObj:=wPaper;
    MoveL Offs(pOrigin,188.59,170.11,0.00),v40,z0,tPen\WObj:=wPaper;
    MoveL Offs(pOrigin,188.59,177.34,0.00),v40,z0,tPen\WObj:=wPaper;
  ENDPROC

  PROC DrawPart45()
    MoveL Offs(pOrigin,188.59,177.34,0.00),v40,z0,tPen\WObj:=wPaper;
    MoveL Offs(pOrigin,189.23,177.76,0.00),v40,z0,tPen\WObj:=wPaper;
    MoveL Offs(pOrigin,189.01,179.04,0.00),v40,z0,tPen\WObj:=wPaper;
    MoveL Offs(pOrigin,189.01,179.04,0.00),v40,z0,tPen\WObj:=wPaper;
    MoveL Offs(pOrigin,189.44,179.46,0.00),v40,z0,tPen\WObj:=wPaper;
    MoveL Offs(pOrigin,189.44,180.31,0.00),v40,z0,tPen\WObj:=wPaper;
    MoveL Offs(pOrigin,189.01,180.52,0.00),v40,z0,tPen\WObj:=wPaper;
    MoveL Offs(pOrigin,189.01,180.52,0.00),v40,z0,tPen\WObj:=wPaper;
    MoveL Offs(pOrigin,188.59,180.10,0.00),v40,z0,tPen\WObj:=wPaper;
    MoveL Offs(pOrigin,188.59,179.25,0.00),v40,z0,tPen\WObj:=wPaper;
    MoveL Offs(pOrigin,189.01,179.04,0.00),v40,z0,tPen\WObj:=wPaper;
    MoveL Offs(pOrigin,188.59,179.04,0.00),v40,z0,tPen\WObj:=wPaper;
    MoveL Offs(pOrigin,188.38,177.55,0.00),v40,z0,tPen\WObj:=wPaper;
    MoveL Offs(pOrigin,188.59,177.34,0.00),v40,z0,tPen\WObj:=wPaper;
    MoveL Offs(pOrigin,188.35,176.70,0.00),v40,z0,tPen\WObj:=wPaper;
    MoveL Offs(pOrigin,189.25,177.60,0.00),v40,z0,tPen\WObj:=wPaper;
    MoveL Offs(pOrigin,189.83,177.79,0.00),v40,z0,tPen\WObj:=wPaper;
    MoveL Offs(pOrigin,187.88,179.75,0.00),v40,z0,tPen\WObj:=wPaper;
    MoveL Offs(pOrigin,188.51,179.84,0.00),v40,z0,tPen\WObj:=wPaper;
    MoveL Offs(pOrigin,189.71,181.04,0.00),v40,z0,tPen\WObj:=wPaper;
    MoveL Offs(pOrigin,189.23,181.38,0.00),v40,z0,tPen\WObj:=wPaper;
    MoveL Offs(pOrigin,189.01,182.23,0.00),v40,z0,tPen\WObj:=wPaper;
    MoveL Offs(pOrigin,189.23,182.44,0.00),v40,z0,tPen\WObj:=wPaper;
    MoveL Offs(pOrigin,189.23,182.44,0.00),v40,z0,tPen\WObj:=wPaper;
    MoveL Offs(pOrigin,189.37,183.29,0.00),v40,z0,tPen\WObj:=wPaper;
    MoveL Offs(pOrigin,189.93,183.93,0.00),v40,z0,tPen\WObj:=wPaper;
    MoveL Offs(pOrigin,192.34,189.24,0.00),v40,z0,tPen\WObj:=wPaper;
    MoveL Offs(pOrigin,194.75,192.64,0.00),v40,z0,tPen\WObj:=wPaper;
    MoveL Offs(pOrigin,198.15,196.25,0.00),v40,z0,tPen\WObj:=wPaper;
    MoveL Offs(pOrigin,202.19,199.65,0.00),v40,z0,tPen\WObj:=wPaper;
    MoveL Offs(pOrigin,202.80,199.17,0.00),v40,z0,tPen\WObj:=wPaper;
    MoveL Offs(pOrigin,205.21,196.77,0.00),v40,z0,tPen\WObj:=wPaper;
    MoveL Offs(pOrigin,204.31,196.17,0.00),v40,z0,tPen\WObj:=wPaper;
    MoveL Offs(pOrigin,201.90,198.58,0.00),v40,fine,tPen\WObj:=wPaper;
    MoveL Offs(pOrigin,201.90,198.58,6.00),v60,z5,tPen\WObj:=wPaper;
    MoveL Offs(pOrigin,203.04,197.69,6.00),vTravel,z5,tPen\WObj:=wPaper;
    MoveL Offs(pOrigin,203.04,197.69,0.00),v60,z0,tPen\WObj:=wPaper;
    MoveL Offs(pOrigin,204.52,197.69,0.00),v40,z0,tPen\WObj:=wPaper;
    MoveL Offs(pOrigin,205.16,198.16,0.00),v40,z0,tPen\WObj:=wPaper;
    MoveL Offs(pOrigin,206.01,199.01,0.00),v40,z0,tPen\WObj:=wPaper;
    MoveL Offs(pOrigin,205.16,198.16,0.00),v40,z0,tPen\WObj:=wPaper;
    MoveL Offs(pOrigin,205.59,198.74,0.00),v40,z0,tPen\WObj:=wPaper;
    MoveL Offs(pOrigin,203.89,198.74,0.00),v40,z0,tPen\WObj:=wPaper;
    MoveL Offs(pOrigin,203.68,198.80,0.00),v40,z0,tPen\WObj:=wPaper;
    MoveL Offs(pOrigin,204.31,199.44,0.00),v40,z0,tPen\WObj:=wPaper;
    MoveL Offs(pOrigin,203.68,198.80,0.00),v40,z0,tPen\WObj:=wPaper;
    MoveL Offs(pOrigin,204.00,199.81,0.00),v40,z0,tPen\WObj:=wPaper;
    MoveL Offs(pOrigin,218.58,214.39,0.00),v40,z0,tPen\WObj:=wPaper;
    MoveL Offs(pOrigin,217.70,214.58,0.00),v40,z0,tPen\WObj:=wPaper;
    MoveL Offs(pOrigin,215.58,214.58,0.00),v40,z0,tPen\WObj:=wPaper;
    MoveL Offs(pOrigin,215.15,215.16,0.00),v40,z0,tPen\WObj:=wPaper;
    MoveL Offs(pOrigin,213.88,216.44,0.00),v40,z0,tPen\WObj:=wPaper;
    MoveL Offs(pOrigin,215.15,215.16,0.00),v40,z0,tPen\WObj:=wPaper;
    MoveL Offs(pOrigin,214.68,214.98,0.00),v40,z0,tPen\WObj:=wPaper;
    MoveL Offs(pOrigin,216.19,216.48,0.00),v40,z0,tPen\WObj:=wPaper;
    MoveL Offs(pOrigin,215.36,216.70,0.00),v40,z0,tPen\WObj:=wPaper;
    MoveL Offs(pOrigin,213.88,216.70,0.00),v40,z0,tPen\WObj:=wPaper;
    MoveL Offs(pOrigin,213.66,216.86,0.00),v40,z0,tPen\WObj:=wPaper;
    MoveL Offs(pOrigin,212.60,217.93,0.00),v40,z0,tPen\WObj:=wPaper;
    MoveL Offs(pOrigin,213.66,216.86,0.00),v40,z0,tPen\WObj:=wPaper;
    MoveL Offs(pOrigin,213.49,216.77,0.00),v40,z0,tPen\WObj:=wPaper;
    MoveL Offs(pOrigin,214.84,218.12,0.00),v40,z0,tPen\WObj:=wPaper;
    MoveL Offs(pOrigin,214.73,217.71,0.00),v40,z0,tPen\WObj:=wPaper;
    MoveL Offs(pOrigin,213.88,218.56,0.00),v40,z0,tPen\WObj:=wPaper;
    MoveL Offs(pOrigin,214.73,217.71,0.00),v40,z0,tPen\WObj:=wPaper;
    MoveL Offs(pOrigin,214.30,217.75,0.00),v40,z0,tPen\WObj:=wPaper;
    MoveL Offs(pOrigin,213.02,217.75,0.00),v40,z0,tPen\WObj:=wPaper;
    MoveL Offs(pOrigin,212.59,217.37,0.00),v40,z0,tPen\WObj:=wPaper;
    MoveL Offs(pOrigin,214.25,219.02,0.00),v40,z0,tPen\WObj:=wPaper;
    MoveL Offs(pOrigin,213.45,218.81,0.00),v40,z0,tPen\WObj:=wPaper;
    MoveL Offs(pOrigin,212.18,218.81,0.00),v40,z0,tPen\WObj:=wPaper;
    MoveL Offs(pOrigin,212.39,218.35,0.00),v40,z0,tPen\WObj:=wPaper;
    MoveL Offs(pOrigin,211.96,218.77,0.00),v40,z0,tPen\WObj:=wPaper;
    MoveL Offs(pOrigin,212.39,218.35,0.00),v40,z0,tPen\WObj:=wPaper;
    MoveL Offs(pOrigin,212.00,218.26,0.00),v40,z0,tPen\WObj:=wPaper;
    MoveL Offs(pOrigin,213.50,219.77,0.00),v40,z0,tPen\WObj:=wPaper;
    MoveL Offs(pOrigin,212.81,219.86,0.00),v40,z0,tPen\WObj:=wPaper;
    MoveL Offs(pOrigin,211.54,219.86,0.00),v40,z0,tPen\WObj:=wPaper;
    MoveL Offs(pOrigin,210.95,220.21,0.00),v40,z0,tPen\WObj:=wPaper;
    MoveL Offs(pOrigin,212.31,221.56,0.00),v40,z0,tPen\WObj:=wPaper;
    MoveL Offs(pOrigin,211.96,220.92,0.00),v40,z0,tPen\WObj:=wPaper;
    MoveL Offs(pOrigin,210.90,220.92,0.00),v40,z0,tPen\WObj:=wPaper;
    MoveL Offs(pOrigin,210.36,221.10,0.00),v40,z0,tPen\WObj:=wPaper;
    MoveL Offs(pOrigin,211.86,222.61,0.00),v40,z0,tPen\WObj:=wPaper;
    MoveL Offs(pOrigin,211.54,222.18,0.00),v40,z0,tPen\WObj:=wPaper;
    MoveL Offs(pOrigin,211.32,222.60,0.00),v40,z0,tPen\WObj:=wPaper;
    MoveL Offs(pOrigin,211.54,222.18,0.00),v40,z0,tPen\WObj:=wPaper;
    MoveL Offs(pOrigin,211.54,221.98,0.00),v40,z0,tPen\WObj:=wPaper;
    MoveL Offs(pOrigin,210.26,221.98,0.00),v40,z0,tPen\WObj:=wPaper;
    MoveL Offs(pOrigin,209.76,222.00,0.00),v40,z0,tPen\WObj:=wPaper;
    MoveL Offs(pOrigin,211.26,223.50,0.00),v40,z0,tPen\WObj:=wPaper;
    MoveL Offs(pOrigin,211.11,223.02,0.00),v40,z0,tPen\WObj:=wPaper;
    MoveL Offs(pOrigin,210.90,223.45,0.00),v40,z0,tPen\WObj:=wPaper;
    MoveL Offs(pOrigin,211.11,223.02,0.00),v40,z0,tPen\WObj:=wPaper;
    MoveL Offs(pOrigin,210.90,223.03,0.00),v40,z0,tPen\WObj:=wPaper;
    MoveL Offs(pOrigin,209.84,223.03,0.00),v40,z0,tPen\WObj:=wPaper;
    MoveL Offs(pOrigin,209.31,223.05,0.00),v40,z0,tPen\WObj:=wPaper;
    MoveL Offs(pOrigin,210.82,224.55,0.00),v40,z0,tPen\WObj:=wPaper;
    MoveL Offs(pOrigin,210.48,224.30,0.00),v40,z0,tPen\WObj:=wPaper;
    MoveL Offs(pOrigin,210.26,224.73,0.00),v40,z0,tPen\WObj:=wPaper;
    MoveL Offs(pOrigin,210.48,224.30,0.00),v40,z0,tPen\WObj:=wPaper;
    MoveL Offs(pOrigin,210.48,224.09,0.00),v40,z0,tPen\WObj:=wPaper;
    MoveL Offs(pOrigin,209.41,224.09,0.00),v40,z0,tPen\WObj:=wPaper;
    MoveL Offs(pOrigin,208.87,224.10,0.00),v40,z0,tPen\WObj:=wPaper;
    MoveL Offs(pOrigin,210.37,225.60,0.00),v40,z0,tPen\WObj:=wPaper;
    MoveL Offs(pOrigin,210.81,225.52,0.00),v40,z0,tPen\WObj:=wPaper;
    MoveL Offs(pOrigin,206.30,230.02,0.00),v40,z0,tPen\WObj:=wPaper;
    MoveL Offs(pOrigin,205.29,229.48,0.00),v40,z0,tPen\WObj:=wPaper;
    MoveL Offs(pOrigin,203.94,228.12,0.00),v40,z0,tPen\WObj:=wPaper;
    MoveL Offs(pOrigin,204.31,228.31,0.00),v40,z0,tPen\WObj:=wPaper;
    MoveL Offs(pOrigin,208.99,228.31,0.00),v40,z0,tPen\WObj:=wPaper;
    MoveL Offs(pOrigin,209.18,228.89,0.00),v40,z0,tPen\WObj:=wPaper;
    MoveL Offs(pOrigin,206.93,226.64,0.00),v40,z0,tPen\WObj:=wPaper;
    MoveL Offs(pOrigin,207.83,226.04,0.00),v40,z0,tPen\WObj:=wPaper;
    MoveL Offs(pOrigin,209.63,227.84,0.00),v40,z0,tPen\WObj:=wPaper;
    MoveL Offs(pOrigin,209.90,227.91,0.00),v40,z0,tPen\WObj:=wPaper;
    MoveL Offs(pOrigin,206.30,231.52,0.00),v40,z0,tPen\WObj:=wPaper;
    MoveL Offs(pOrigin,206.94,231.13,0.00),v40,z0,tPen\WObj:=wPaper;
    MoveL Offs(pOrigin,208.14,232.33,0.00),v40,z0,tPen\WObj:=wPaper;
    MoveL Offs(pOrigin,207.93,232.38,0.00),v40,z0,tPen\WObj:=wPaper;
  ENDPROC

  PROC DrawPart46()
    MoveL Offs(pOrigin,207.93,233.23,0.00),v40,z0,tPen\WObj:=wPaper;
    MoveL Offs(pOrigin,207.29,233.65,0.00),v40,z0,tPen\WObj:=wPaper;
    MoveL Offs(pOrigin,207.29,233.65,0.00),v40,z0,tPen\WObj:=wPaper;
    MoveL Offs(pOrigin,206.65,241.51,0.00),v40,z0,tPen\WObj:=wPaper;
    MoveL Offs(pOrigin,206.65,241.51,0.00),v40,z0,tPen\WObj:=wPaper;
    MoveL Offs(pOrigin,205.80,241.94,0.00),v40,z0,tPen\WObj:=wPaper;
    MoveL Offs(pOrigin,205.59,243.21,0.00),v40,z0,tPen\WObj:=wPaper;
    MoveL Offs(pOrigin,205.59,243.21,0.00),v40,z0,tPen\WObj:=wPaper;
    MoveL Offs(pOrigin,205.09,243.85,0.00),v40,z0,tPen\WObj:=wPaper;
    MoveL Offs(pOrigin,204.81,245.34,0.00),v40,z0,tPen\WObj:=wPaper;
    MoveL Offs(pOrigin,204.95,247.04,0.00),v40,z0,tPen\WObj:=wPaper;
    MoveL Offs(pOrigin,205.59,248.10,0.00),v40,z0,tPen\WObj:=wPaper;
    MoveL Offs(pOrigin,205.50,247.60,0.00),v40,z0,tPen\WObj:=wPaper;
    MoveL Offs(pOrigin,207.30,249.41,0.00),v40,z0,tPen\WObj:=wPaper;
    MoveL Offs(pOrigin,206.86,249.43,0.00),v40,z0,tPen\WObj:=wPaper;
    MoveL Offs(pOrigin,205.59,249.43,0.00),v40,z0,tPen\WObj:=wPaper;
    MoveL Offs(pOrigin,205.38,250.23,0.00),v40,z0,tPen\WObj:=wPaper;
    MoveL Offs(pOrigin,205.66,248.31,0.00),v40,z0,tPen\WObj:=wPaper;
    MoveL Offs(pOrigin,206.44,248.17,0.00),v40,z0,tPen\WObj:=wPaper;
    MoveL Offs(pOrigin,207.07,248.95,0.00),v40,z0,tPen\WObj:=wPaper;
    MoveL Offs(pOrigin,207.29,251.71,0.00),v40,z0,tPen\WObj:=wPaper;
    MoveL Offs(pOrigin,207.07,257.02,0.00),v40,z0,tPen\WObj:=wPaper;
    MoveL Offs(pOrigin,208.07,258.30,0.00),v40,z0,tPen\WObj:=wPaper;
    MoveL Offs(pOrigin,207.93,258.94,0.00),v40,z0,tPen\WObj:=wPaper;
    MoveL Offs(pOrigin,207.93,258.94,0.00),v40,z0,tPen\WObj:=wPaper;
    MoveL Offs(pOrigin,207.93,260.00,0.00),v40,z0,tPen\WObj:=wPaper;
    MoveL Offs(pOrigin,207.29,260.85,0.00),v40,z0,tPen\WObj:=wPaper;
    MoveL Offs(pOrigin,207.33,261.39,0.00),v40,z0,tPen\WObj:=wPaper;
    MoveL Offs(pOrigin,202.83,256.88,0.00),v40,z0,tPen\WObj:=wPaper;
    MoveL Offs(pOrigin,203.46,256.82,0.00),v40,z0,tPen\WObj:=wPaper;
    MoveL Offs(pOrigin,207.29,256.82,0.00),v40,z0,tPen\WObj:=wPaper;
    MoveL Offs(pOrigin,207.29,257.24,0.00),v40,z0,tPen\WObj:=wPaper;
    MoveL Offs(pOrigin,207.71,257.45,0.00),v40,z0,tPen\WObj:=wPaper;
    MoveL Offs(pOrigin,208.07,257.24,0.00),v40,z0,tPen\WObj:=wPaper;
    MoveL Offs(pOrigin,209.34,253.41,0.00),v40,z0,tPen\WObj:=wPaper;
    MoveL Offs(pOrigin,210.90,251.07,0.00),v40,z0,tPen\WObj:=wPaper;
    MoveL Offs(pOrigin,211.96,250.30,0.00),v40,z0,tPen\WObj:=wPaper;
    MoveL Offs(pOrigin,214.94,249.59,0.00),v40,z0,tPen\WObj:=wPaper;
    MoveL Offs(pOrigin,223.65,249.80,0.00),v40,z0,tPen\WObj:=wPaper;
    MoveL Offs(pOrigin,230.45,251.07,0.00),v40,z0,tPen\WObj:=wPaper;
    MoveL Offs(pOrigin,232.79,251.85,0.00),v40,z0,tPen\WObj:=wPaper;
    MoveL Offs(pOrigin,234.91,253.62,0.00),v40,z0,tPen\WObj:=wPaper;
    MoveL Offs(pOrigin,235.55,254.90,0.00),v40,z0,tPen\WObj:=wPaper;
    MoveL Offs(pOrigin,234.58,254.28,0.00),v40,z0,tPen\WObj:=wPaper;
    MoveL Offs(pOrigin,238.03,257.74,0.00),v40,z0,tPen\WObj:=wPaper;
    MoveL Offs(pOrigin,238.57,257.49,0.00),v40,z0,tPen\WObj:=wPaper;
    MoveL Offs(pOrigin,224.00,272.06,0.00),v40,z0,tPen\WObj:=wPaper;
    MoveL Offs(pOrigin,223.39,271.48,0.00),v40,z0,tPen\WObj:=wPaper;
    MoveL Offs(pOrigin,217.68,265.77,0.00),v40,z0,tPen\WObj:=wPaper;
    MoveL Offs(pOrigin,217.70,266.33,0.00),v40,z0,tPen\WObj:=wPaper;
    MoveL Offs(pOrigin,214.72,266.33,0.00),v40,fine,tPen\WObj:=wPaper;
    MoveL Offs(pOrigin,214.72,266.33,6.00),v60,z5,tPen\WObj:=wPaper;
    MoveL Offs(pOrigin,215.36,265.27,6.00),vTravel,z5,tPen\WObj:=wPaper;
    MoveL Offs(pOrigin,215.36,265.27,0.00),v60,z0,tPen\WObj:=wPaper;
    MoveL Offs(pOrigin,213.88,265.27,0.00),v40,z0,tPen\WObj:=wPaper;
    MoveL Offs(pOrigin,213.04,265.60,0.00),v40,z0,tPen\WObj:=wPaper;
    MoveL Offs(pOrigin,218.30,270.86,0.00),v40,z0,tPen\WObj:=wPaper;
    MoveL Offs(pOrigin,218.91,271.18,0.00),v40,z0,tPen\WObj:=wPaper;
    MoveL Offs(pOrigin,232.88,257.20,0.00),v40,z0,tPen\WObj:=wPaper;
    MoveL Offs(pOrigin,232.14,256.46,0.00),v40,z0,tPen\WObj:=wPaper;
    MoveL Offs(pOrigin,217.56,271.03,0.00),v40,z0,tPen\WObj:=wPaper;
    MoveL Offs(pOrigin,217.27,271.05,0.00),v40,z0,tPen\WObj:=wPaper;
    MoveL Offs(pOrigin,217.13,270.62,0.00),v40,z0,tPen\WObj:=wPaper;
    MoveL Offs(pOrigin,217.49,270.41,0.00),v40,z0,tPen\WObj:=wPaper;
    MoveL Offs(pOrigin,226.41,271.69,0.00),v40,z0,tPen\WObj:=wPaper;
    MoveL Offs(pOrigin,230.88,271.26,0.00),v40,z0,tPen\WObj:=wPaper;
    MoveL Offs(pOrigin,231.73,271.90,0.00),v40,z0,tPen\WObj:=wPaper;
    MoveL Offs(pOrigin,231.18,271.80,0.00),v40,z0,tPen\WObj:=wPaper;
    MoveL Offs(pOrigin,219.16,259.78,0.00),v40,z0,tPen\WObj:=wPaper;
    MoveL Offs(pOrigin,219.82,260.00,0.00),v40,z0,tPen\WObj:=wPaper;
    MoveL Offs(pOrigin,219.82,260.64,0.00),v40,z0,tPen\WObj:=wPaper;
    MoveL Offs(pOrigin,220.68,260.64,0.00),v40,z0,tPen\WObj:=wPaper;
    MoveL Offs(pOrigin,220.68,260.64,0.00),v40,z0,tPen\WObj:=wPaper;
    MoveL Offs(pOrigin,220.46,259.79,0.00),v40,z0,tPen\WObj:=wPaper;
    MoveL Offs(pOrigin,219.82,260.00,0.00),v40,z0,tPen\WObj:=wPaper;
    MoveL Offs(pOrigin,219.82,260.00,0.00),v40,z0,tPen\WObj:=wPaper;
    MoveL Offs(pOrigin,218.55,259.93,0.00),v40,z0,tPen\WObj:=wPaper;
    MoveL Offs(pOrigin,217.27,259.15,0.00),v40,z0,tPen\WObj:=wPaper;
    MoveL Offs(pOrigin,216.21,259.58,0.00),v40,z0,tPen\WObj:=wPaper;
    MoveL Offs(pOrigin,216.21,259.58,0.00),v40,z0,tPen\WObj:=wPaper;
    MoveL Offs(pOrigin,217.06,261.49,0.00),v40,z0,tPen\WObj:=wPaper;
    MoveL Offs(pOrigin,218.34,262.12,0.00),v40,z0,tPen\WObj:=wPaper;
    MoveL Offs(pOrigin,218.34,262.12,0.00),v40,z0,tPen\WObj:=wPaper;
    MoveL Offs(pOrigin,218.76,262.76,0.00),v40,z0,tPen\WObj:=wPaper;
    MoveL Offs(pOrigin,220.46,263.90,0.00),v40,z0,tPen\WObj:=wPaper;
    MoveL Offs(pOrigin,222.38,264.75,0.00),v40,z0,tPen\WObj:=wPaper;
    MoveL Offs(pOrigin,228.11,266.59,0.00),v40,z0,tPen\WObj:=wPaper;
    MoveL Offs(pOrigin,229.18,266.59,0.00),v40,z0,tPen\WObj:=wPaper;
    MoveL Offs(pOrigin,229.81,267.01,0.00),v40,z0,tPen\WObj:=wPaper;
    MoveL Offs(pOrigin,229.81,267.01,0.00),v40,z0,tPen\WObj:=wPaper;
    MoveL Offs(pOrigin,229.18,267.65,0.00),v40,z0,tPen\WObj:=wPaper;
    MoveL Offs(pOrigin,229.18,267.65,0.00),v40,z0,tPen\WObj:=wPaper;
    MoveL Offs(pOrigin,229.60,268.50,0.00),v40,z0,tPen\WObj:=wPaper;
    MoveL Offs(pOrigin,230.45,268.71,0.00),v40,z0,tPen\WObj:=wPaper;
    MoveL Offs(pOrigin,230.45,268.71,0.00),v40,z0,tPen\WObj:=wPaper;
    MoveL Offs(pOrigin,231.65,269.77,0.00),v40,z0,tPen\WObj:=wPaper;
    MoveL Offs(pOrigin,231.51,270.84,0.00),v40,z0,tPen\WObj:=wPaper;
    MoveL Offs(pOrigin,231.51,270.84,0.00),v40,z0,tPen\WObj:=wPaper;
    MoveL Offs(pOrigin,233.21,270.84,0.00),v40,z0,tPen\WObj:=wPaper;
    MoveL Offs(pOrigin,233.21,270.84,0.00),v40,z0,tPen\WObj:=wPaper;
    MoveL Offs(pOrigin,233.00,268.57,0.00),v40,z0,tPen\WObj:=wPaper;
    MoveL Offs(pOrigin,234.06,268.29,0.00),v40,z0,tPen\WObj:=wPaper;
    MoveL Offs(pOrigin,235.48,269.14,0.00),v40,z0,tPen\WObj:=wPaper;
    MoveL Offs(pOrigin,236.19,271.90,0.00),v40,z0,tPen\WObj:=wPaper;
    MoveL Offs(pOrigin,236.19,275.30,0.00),v40,fine,tPen\WObj:=wPaper;
    MoveL Offs(pOrigin,236.19,275.30,6.00),v60,z5,tPen\WObj:=wPaper;
    MoveL Offs(pOrigin,235.98,273.52,6.00),vTravel,z5,tPen\WObj:=wPaper;
    MoveL Offs(pOrigin,235.98,273.52,0.00),v60,z0,tPen\WObj:=wPaper;
    MoveL Offs(pOrigin,236.88,272.62,0.00),v40,fine,tPen\WObj:=wPaper;
    MoveL Offs(pOrigin,236.88,272.62,6.00),v60,z5,tPen\WObj:=wPaper;
    MoveL Offs(pOrigin,236.19,271.48,6.00),vTravel,z5,tPen\WObj:=wPaper;
    MoveL Offs(pOrigin,236.19,271.48,0.00),v60,z0,tPen\WObj:=wPaper;
    MoveL Offs(pOrigin,236.61,271.05,0.00),v40,z0,tPen\WObj:=wPaper;
    MoveL Offs(pOrigin,236.40,267.86,0.00),v40,z0,tPen\WObj:=wPaper;
    MoveL Offs(pOrigin,237.46,267.15,0.00),v40,z0,tPen\WObj:=wPaper;
    MoveL Offs(pOrigin,241.50,267.86,0.00),v40,z0,tPen\WObj:=wPaper;
    MoveL Offs(pOrigin,244.26,267.86,0.00),v40,z0,tPen\WObj:=wPaper;
    MoveL Offs(pOrigin,245.32,268.92,0.00),v40,z0,tPen\WObj:=wPaper;
    MoveL Offs(pOrigin,245.32,268.92,0.00),v40,z0,tPen\WObj:=wPaper;
    MoveL Offs(pOrigin,245.11,269.77,0.00),v40,z0,tPen\WObj:=wPaper;
  ENDPROC

  PROC DrawPart47()
    MoveL Offs(pOrigin,245.32,270.13,0.00),v40,z0,tPen\WObj:=wPaper;
    MoveL Offs(pOrigin,246.81,270.20,0.00),v40,z0,tPen\WObj:=wPaper;
    MoveL Offs(pOrigin,246.81,270.20,0.00),v40,z0,tPen\WObj:=wPaper;
    MoveL Offs(pOrigin,246.81,269.14,0.00),v40,z0,tPen\WObj:=wPaper;
    MoveL Offs(pOrigin,246.81,269.14,0.00),v40,z0,tPen\WObj:=wPaper;
    MoveL Offs(pOrigin,246.60,267.86,0.00),v40,z0,tPen\WObj:=wPaper;
    MoveL Offs(pOrigin,246.60,267.86,0.00),v40,z0,tPen\WObj:=wPaper;
    MoveL Offs(pOrigin,245.96,267.93,0.00),v40,z0,tPen\WObj:=wPaper;
    MoveL Offs(pOrigin,245.75,268.50,0.00),v40,z0,tPen\WObj:=wPaper;
    MoveL Offs(pOrigin,246.81,269.14,0.00),v40,fine,tPen\WObj:=wPaper;
    MoveL Offs(pOrigin,246.81,269.14,6.00),v60,z5,tPen\WObj:=wPaper;
    MoveL Offs(pOrigin,246.60,267.86,6.00),vTravel,z5,tPen\WObj:=wPaper;
    MoveL Offs(pOrigin,246.60,267.86,0.00),v60,z0,tPen\WObj:=wPaper;
    MoveL Offs(pOrigin,246.39,266.02,0.00),v40,z0,tPen\WObj:=wPaper;
    MoveL Offs(pOrigin,244.69,266.16,0.00),v40,z0,tPen\WObj:=wPaper;
    MoveL Offs(pOrigin,244.69,266.16,0.00),v40,z0,tPen\WObj:=wPaper;
    MoveL Offs(pOrigin,245.32,264.89,0.00),v40,z0,tPen\WObj:=wPaper;
    MoveL Offs(pOrigin,245.32,264.89,0.00),v40,z0,tPen\WObj:=wPaper;
    MoveL Offs(pOrigin,245.11,263.61,0.00),v40,z0,tPen\WObj:=wPaper;
    MoveL Offs(pOrigin,246.46,260.07,0.00),v40,z0,tPen\WObj:=wPaper;
    MoveL Offs(pOrigin,247.88,258.16,0.00),v40,z0,tPen\WObj:=wPaper;
    MoveL Offs(pOrigin,249.15,257.88,0.00),v40,z0,tPen\WObj:=wPaper;
    MoveL Offs(pOrigin,249.15,257.88,0.00),v40,z0,tPen\WObj:=wPaper;
    MoveL Offs(pOrigin,249.36,257.02,0.00),v40,z0,tPen\WObj:=wPaper;
    MoveL Offs(pOrigin,251.91,254.83,0.00),v40,z0,tPen\WObj:=wPaper;
    MoveL Offs(pOrigin,256.16,254.05,0.00),v40,z0,tPen\WObj:=wPaper;
    MoveL Offs(pOrigin,259.56,254.05,0.00),v40,z0,tPen\WObj:=wPaper;
    MoveL Offs(pOrigin,265.09,254.69,0.00),v40,z0,tPen\WObj:=wPaper;
    MoveL Offs(pOrigin,269.12,255.54,0.00),v40,z0,tPen\WObj:=wPaper;
    MoveL Offs(pOrigin,273.16,256.88,0.00),v40,z0,tPen\WObj:=wPaper;
    MoveL Offs(pOrigin,274.86,258.09,0.00),v40,z0,tPen\WObj:=wPaper;
    MoveL Offs(pOrigin,276.49,261.06,0.00),v40,z0,tPen\WObj:=wPaper;
    MoveL Offs(pOrigin,276.28,262.12,0.00),v40,z0,tPen\WObj:=wPaper;
    MoveL Offs(pOrigin,276.77,263.40,0.00),v40,z0,tPen\WObj:=wPaper;
    MoveL Offs(pOrigin,276.35,264.25,0.00),v40,z0,tPen\WObj:=wPaper;
    MoveL Offs(pOrigin,276.35,266.16,0.00),v40,z0,tPen\WObj:=wPaper;
    MoveL Offs(pOrigin,276.85,267.86,0.00),v40,z0,tPen\WObj:=wPaper;
    MoveL Offs(pOrigin,279.33,269.21,0.00),v40,z0,tPen\WObj:=wPaper;
    MoveL Offs(pOrigin,280.39,271.05,0.00),v40,z0,tPen\WObj:=wPaper;
    MoveL Offs(pOrigin,280.39,271.05,0.00),v40,z0,tPen\WObj:=wPaper;
    MoveL Offs(pOrigin,282.30,271.33,0.00),v40,z0,tPen\WObj:=wPaper;
    MoveL Offs(pOrigin,283.15,272.33,0.00),v40,z0,tPen\WObj:=wPaper;
    MoveL Offs(pOrigin,283.15,272.33,0.00),v40,z0,tPen\WObj:=wPaper;
    MoveL Offs(pOrigin,283.15,272.11,0.00),v40,z0,tPen\WObj:=wPaper;
    MoveL Offs(pOrigin,284.00,272.33,0.00),v40,z0,tPen\WObj:=wPaper;
    MoveL Offs(pOrigin,284.00,272.33,0.00),v40,z0,tPen\WObj:=wPaper;
    MoveL Offs(pOrigin,284.64,272.96,0.00),v40,z0,tPen\WObj:=wPaper;
    MoveL Offs(pOrigin,285.70,272.96,0.00),v40,z0,tPen\WObj:=wPaper;
    MoveL Offs(pOrigin,286.55,272.33,0.00),v40,z0,tPen\WObj:=wPaper;
    MoveL Offs(pOrigin,286.55,272.33,0.00),v40,z0,tPen\WObj:=wPaper;
    MoveL Offs(pOrigin,286.12,271.69,0.00),v40,z0,tPen\WObj:=wPaper;
    MoveL Offs(pOrigin,285.49,271.69,0.00),v40,z0,tPen\WObj:=wPaper;
    MoveL Offs(pOrigin,285.13,271.26,0.00),v40,z0,tPen\WObj:=wPaper;
    MoveL Offs(pOrigin,285.13,267.22,0.00),v40,z0,tPen\WObj:=wPaper;
    MoveL Offs(pOrigin,284.85,267.38,0.00),v40,z0,tPen\WObj:=wPaper;
    MoveL Offs(pOrigin,289.52,267.38,0.00),v40,z0,tPen\WObj:=wPaper;
    MoveL Offs(pOrigin,290.04,267.94,0.00),v40,z0,tPen\WObj:=wPaper;
    MoveL Offs(pOrigin,285.54,263.43,0.00),v40,z0,tPen\WObj:=wPaper;
    MoveL Offs(pOrigin,286.12,263.16,0.00),v40,z0,tPen\WObj:=wPaper;
    MoveL Offs(pOrigin,289.52,263.16,0.00),v40,z0,tPen\WObj:=wPaper;
    MoveL Offs(pOrigin,289.74,262.76,0.00),v40,z0,tPen\WObj:=wPaper;
    MoveL Offs(pOrigin,290.38,266.16,0.00),v40,z0,tPen\WObj:=wPaper;
    MoveL Offs(pOrigin,290.38,266.16,0.00),v40,z0,tPen\WObj:=wPaper;
    MoveL Offs(pOrigin,290.80,267.01,0.00),v40,z0,tPen\WObj:=wPaper;
    MoveL Offs(pOrigin,291.86,267.65,0.00),v40,z0,tPen\WObj:=wPaper;
    MoveL Offs(pOrigin,294.84,270.62,0.00),v40,z0,tPen\WObj:=wPaper;
    MoveL Offs(pOrigin,294.84,270.62,0.00),v40,z0,tPen\WObj:=wPaper;
    MoveL Offs(pOrigin,295.05,271.26,0.00),v40,z0,tPen\WObj:=wPaper;
    MoveL Offs(pOrigin,296.33,271.69,0.00),v40,z0,tPen\WObj:=wPaper;
    MoveL Offs(pOrigin,297.32,271.40,0.00),v40,z0,tPen\WObj:=wPaper;
    MoveL Offs(pOrigin,299.16,268.50,0.00),v40,z0,tPen\WObj:=wPaper;
    MoveL Offs(pOrigin,299.94,265.10,0.00),v40,z0,tPen\WObj:=wPaper;
    MoveL Offs(pOrigin,299.30,260.64,0.00),v40,z0,tPen\WObj:=wPaper;
    MoveL Offs(pOrigin,298.31,258.94,0.00),v40,z0,tPen\WObj:=wPaper;
    MoveL Offs(pOrigin,298.66,257.24,0.00),v40,z0,tPen\WObj:=wPaper;
    MoveL Offs(pOrigin,298.10,256.39,0.00),v40,z0,tPen\WObj:=wPaper;
    MoveL Offs(pOrigin,296.89,252.14,0.00),v40,z0,tPen\WObj:=wPaper;
    MoveL Offs(pOrigin,295.05,248.95,0.00),v40,z0,tPen\WObj:=wPaper;
    MoveL Offs(pOrigin,295.82,249.52,0.00),v40,z0,tPen\WObj:=wPaper;
    MoveL Offs(pOrigin,295.07,250.27,0.00),v40,fine,tPen\WObj:=wPaper;
    MoveL Offs(pOrigin,295.07,250.27,6.00),v60,z5,tPen\WObj:=wPaper;
    MoveL Offs(pOrigin,295.37,251.47,6.00),vTravel,z5,tPen\WObj:=wPaper;
    MoveL Offs(pOrigin,295.37,251.47,0.00),v60,z0,tPen\WObj:=wPaper;
    MoveL Offs(pOrigin,296.72,250.12,0.00),v40,fine,tPen\WObj:=wPaper;
    MoveL Offs(pOrigin,296.72,250.12,6.00),v60,z5,tPen\WObj:=wPaper;
    MoveL Offs(pOrigin,297.62,249.22,6.00),vTravel,z5,tPen\WObj:=wPaper;
    MoveL Offs(pOrigin,297.62,249.22,0.00),v60,z0,tPen\WObj:=wPaper;
    MoveL Offs(pOrigin,302.58,244.26,0.00),v40,z0,tPen\WObj:=wPaper;
    MoveL Offs(pOrigin,302.86,244.91,0.00),v40,z0,tPen\WObj:=wPaper;
    MoveL Offs(pOrigin,304.66,246.71,0.00),v40,z0,tPen\WObj:=wPaper;
    MoveL Offs(pOrigin,304.07,247.25,0.00),v40,z0,tPen\WObj:=wPaper;
    MoveL Offs(pOrigin,307.07,244.24,0.00),v40,z0,tPen\WObj:=wPaper;
    MoveL Offs(pOrigin,307.35,244.92,0.00),v40,z0,tPen\WObj:=wPaper;
    MoveL Offs(pOrigin,309.15,246.72,0.00),v40,z0,tPen\WObj:=wPaper;
    MoveL Offs(pOrigin,308.56,247.24,0.00),v40,z0,tPen\WObj:=wPaper;
    MoveL Offs(pOrigin,311.57,244.23,0.00),v40,z0,tPen\WObj:=wPaper;
    MoveL Offs(pOrigin,311.84,244.93,0.00),v40,z0,tPen\WObj:=wPaper;
    MoveL Offs(pOrigin,313.65,246.74,0.00),v40,z0,tPen\WObj:=wPaper;
    MoveL Offs(pOrigin,313.06,247.22,0.00),v40,z0,tPen\WObj:=wPaper;
    MoveL Offs(pOrigin,316.06,244.22,0.00),v40,z0,tPen\WObj:=wPaper;
    MoveL Offs(pOrigin,316.19,244.80,0.00),v40,z0,tPen\WObj:=wPaper;
    MoveL Offs(pOrigin,318.14,246.75,0.00),v40,z0,tPen\WObj:=wPaper;
    MoveL Offs(pOrigin,317.70,247.06,0.00),v40,z0,tPen\WObj:=wPaper;
    MoveL Offs(pOrigin,320.86,243.90,0.00),v40,z0,tPen\WObj:=wPaper;
    MoveL Offs(pOrigin,320.68,244.81,0.00),v40,z0,tPen\WObj:=wPaper;
    MoveL Offs(pOrigin,322.33,246.46,0.00),v40,z0,tPen\WObj:=wPaper;
    MoveL Offs(pOrigin,322.49,246.74,0.00),v40,z0,tPen\WObj:=wPaper;
    MoveL Offs(pOrigin,325.50,243.74,0.00),v40,z0,tPen\WObj:=wPaper;
    MoveL Offs(pOrigin,324.88,244.52,0.00),v40,z0,tPen\WObj:=wPaper;
    MoveL Offs(pOrigin,326.68,246.33,0.00),v40,z0,tPen\WObj:=wPaper;
    MoveL Offs(pOrigin,327.14,246.58,0.00),v40,z0,tPen\WObj:=wPaper;
    MoveL Offs(pOrigin,330.14,243.57,0.00),v40,z0,tPen\WObj:=wPaper;
    MoveL Offs(pOrigin,330.42,244.09,0.00),v40,z0,tPen\WObj:=wPaper;
    MoveL Offs(pOrigin,332.22,245.90,0.00),v40,z0,tPen\WObj:=wPaper;
    MoveL Offs(pOrigin,331.93,246.27,0.00),v40,z0,tPen\WObj:=wPaper;
    MoveL Offs(pOrigin,334.94,243.26,0.00),v40,z0,tPen\WObj:=wPaper;
    MoveL Offs(pOrigin,334.76,243.96,0.00),v40,z0,tPen\WObj:=wPaper;
    MoveL Offs(pOrigin,336.56,245.76,0.00),v40,z0,tPen\WObj:=wPaper;
    MoveL Offs(pOrigin,336.73,245.95,0.00),v40,z0,tPen\WObj:=wPaper;
    MoveL Offs(pOrigin,339.88,242.80,0.00),v40,z0,tPen\WObj:=wPaper;
  ENDPROC

